// SIMATIC S7-200 project (STEP 7-Micro/WIN), CPU 224XP CN REL 02.01

SYMBOL_TABLE S7-200 符号
Always_On        SM0.0    // 始终接通为 ON
First_Scan_On    SM0.1    // 仅第一个扫描周期中接通为 ON
Xmit0_Idle       SM4.5    // 当发送器处于空闲状态时（端口 0），置位为 1
P0_Config        SMB30    // 通信端口 0 设置：奇偶校验、每个字符的数据位数目、波特率和协议
P0_Stat_Rcv      SMB86    // 端口 0 信息接收状态
P0_Ctrl_Rcv      SMB87    // 信息接收控制
P0_Start_Char    SMB88    // 信息起始字符
P0_End_Char      SMB89    // 信息结束字符
P0_Max_Char      SMB94    // 信息接收最大字符数（1 至 255 个字节）
P1_Config        SMB130   // 通信端口 1 设置：奇偶校验、每个字符的数据位数目、波特率和协议
P0_Idle_Time     SMW90    // 空闲线时间，以毫秒为单位表示
END_SYMBOL_TABLE

ORGANIZATION_BLOCK 主程序:OB1
TITLE=程序注释
BEGIN
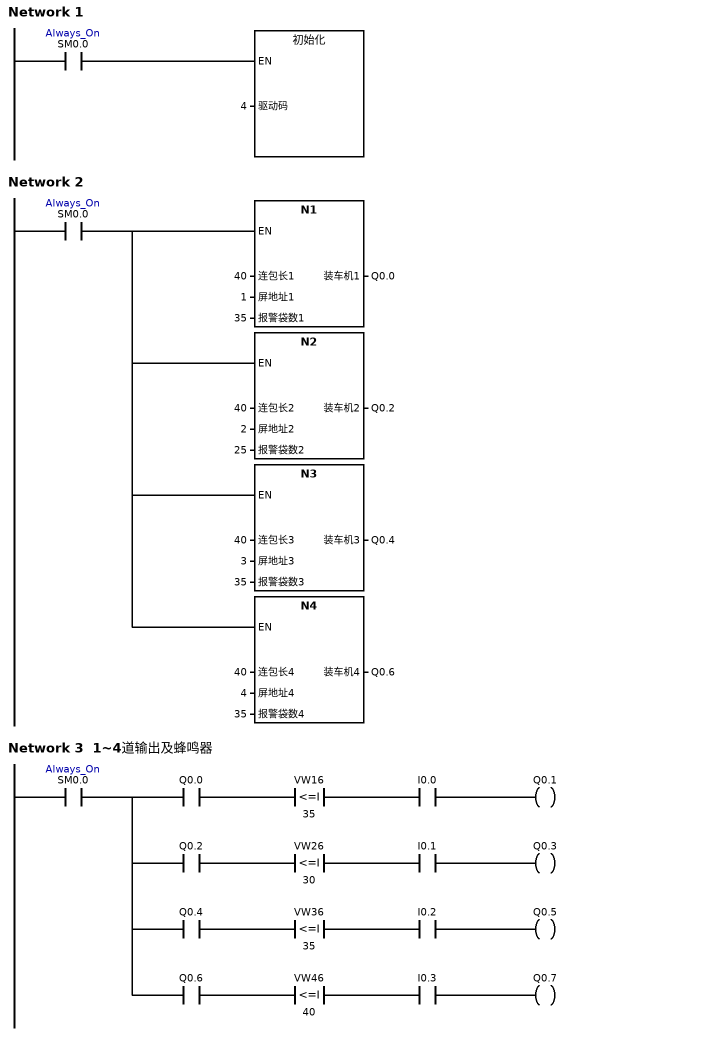
Network 1
LD     Always_On:SM0.0
CALL   初始化:SBR0, 4
Network 2
LD     Always_On:SM0.0
CALL   N1:SBR1, 40, 1, 35, Q0.0
CALL   N2:SBR2, 40, 2, 25, Q0.2
CALL   N3:SBR3, 40, 3, 35, Q0.4
CALL   N4:SBR4, 40, 4, 35, Q0.6
Network 3 // 1~4道输出及蜂鸣器
LD     Always_On:SM0.0
LPS
A      Q0.0
AW<=   VW16, 35
A      I0.0
=      Q0.1
LRD
A      Q0.2
AW<=   VW26, 30
A      I0.1
=      Q0.3
LRD
A      Q0.4
AW<=   VW36, 35
A      I0.2
=      Q0.5
LPP
A      Q0.6
AW<=   VW46, 40
A      I0.3
=      Q0.7
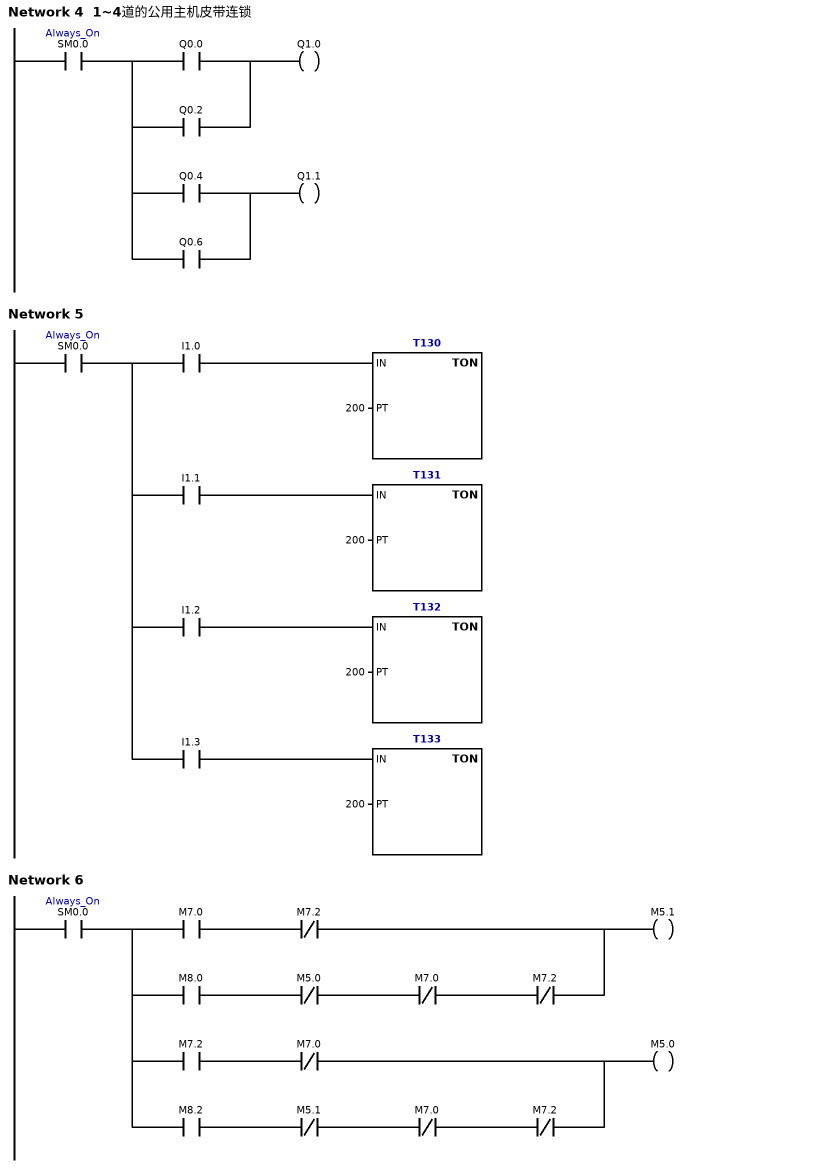
Network 4 // 1~4道的公用主机皮带连锁
LD     Always_On:SM0.0
LPS
LD     Q0.0
O      Q0.2
ALD
=      Q1.0
LPP
LD     Q0.4
O      Q0.6
ALD
=      Q1.1
Network 5
LD     Always_On:SM0.0
LPS
A      I1.0
TON    T130, 200
LRD
A      I1.1
TON    T131, 200
LRD
A      I1.2
TON    T132, 200
LPP
A      I1.3
TON    T133, 200
Network 6
LD     Always_On:SM0.0
LPS
LD     M7.0
AN     M7.2
LD     M8.0
AN     M5.0
AN     M7.0
AN     M7.2
OLD
ALD
=      M5.1
LPP
LD     M7.2
AN     M7.0
LD     M8.2
AN     M5.1
AN     M7.0
AN     M7.2
OLD
ALD
=      M5.0
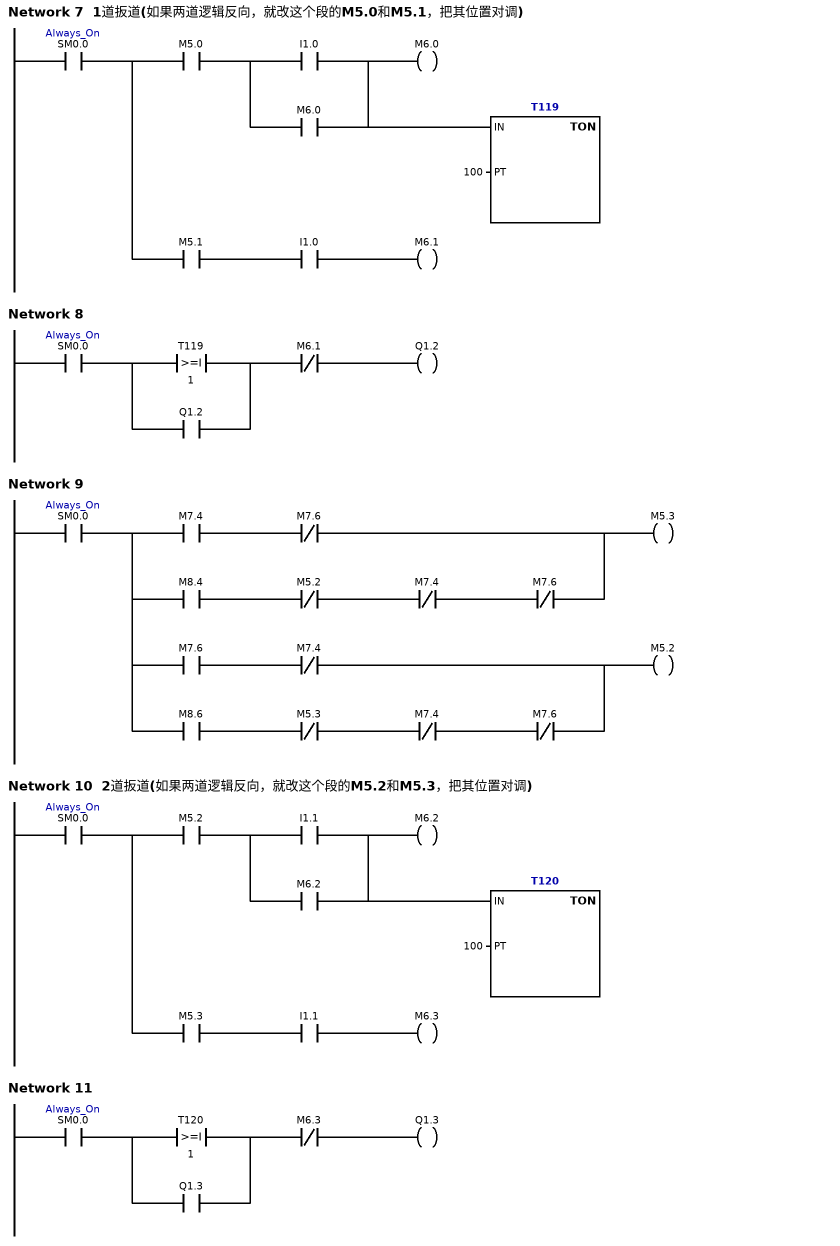
Network 7 // 1道扳道(如果两道逻辑反向，就改这个段的M5.0和M5.1，把其位置对调)
LD     Always_On:SM0.0
LPS
A      M5.0
LD     I1.0
O      M6.0
ALD
=      M6.0
TON    T119, 100
LPP
A      M5.1
A      I1.0
=      M6.1
Network 8
LD     Always_On:SM0.0
LDW>=  T119, 1
O      Q1.2
ALD
AN     M6.1
=      Q1.2
Network 9
LD     Always_On:SM0.0
LPS
LD     M7.4
AN     M7.6
LD     M8.4
AN     M5.2
AN     M7.4
AN     M7.6
OLD
ALD
=      M5.3
LPP
LD     M7.6
AN     M7.4
LD     M8.6
AN     M5.3
AN     M7.4
AN     M7.6
OLD
ALD
=      M5.2
Network 10 // 2道扳道(如果两道逻辑反向，就改这个段的M5.2和M5.3，把其位置对调)
LD     Always_On:SM0.0
LPS
A      M5.2
LD     I1.1
O      M6.2
ALD
=      M6.2
TON    T120, 100
LPP
A      M5.3
A      I1.1
=      M6.3
Network 11
LD     Always_On:SM0.0
LDW>=  T120, 1
O      Q1.3
ALD
AN     M6.3
=      Q1.3
END_ORGANIZATION_BLOCK

SUBROUTINE_BLOCK 初始化:SBR0
TITLE=子程序注释
VAR_INPUT
驱动码:WORD;	// LW0 
END_VAR
VAR
temp1:WORD;	// LW2 
temp2:WORD;	// LW4 
END_VAR
BEGIN
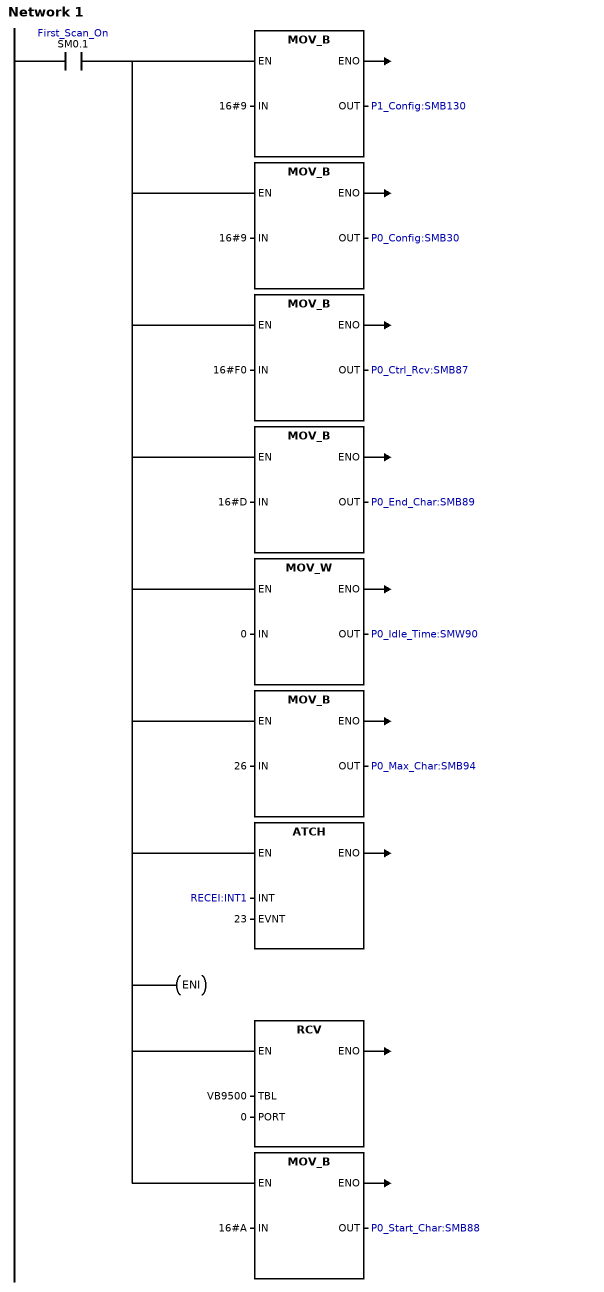
Network 1
// 首次扫描时，
// 初始化自由端口：
// - 选择9600波特
// - 选择8个数据位
// - 选择无校验
// 初始化RCV信息控制字节：
// - RCV被启用
// - 检测到信息字符结束
// - 将空闲行条件检测为
// 信息开始条件。
// 将信息字符结束设为hex OA（换行符）。
// 将空闲行超时设为5毫秒。
// 将最大字符数设为100。
// 为端口0在VB100位置启用带缓冲区的接收方框
LD     First_Scan_On:SM0.1
MOVB   16#9, P1_Config:SMB130
MOVB   16#9, P0_Config:SMB30
MOVB   16#F0, P0_Ctrl_Rcv:SMB87
MOVB   16#D, P0_End_Char:SMB89
MOVW   0, P0_Idle_Time:SMW90
MOVB   26, P0_Max_Char:SMB94
ATCH   RECEI:INT1, 23
ENI
RCV    VB9500, 0
MOVB   16#A, P0_Start_Char:SMB88
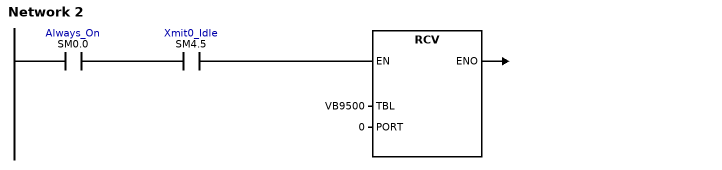
Network 2
LD     Always_On:SM0.0
A      Xmit0_Idle:SM4.5
RCV    VB9500, 0
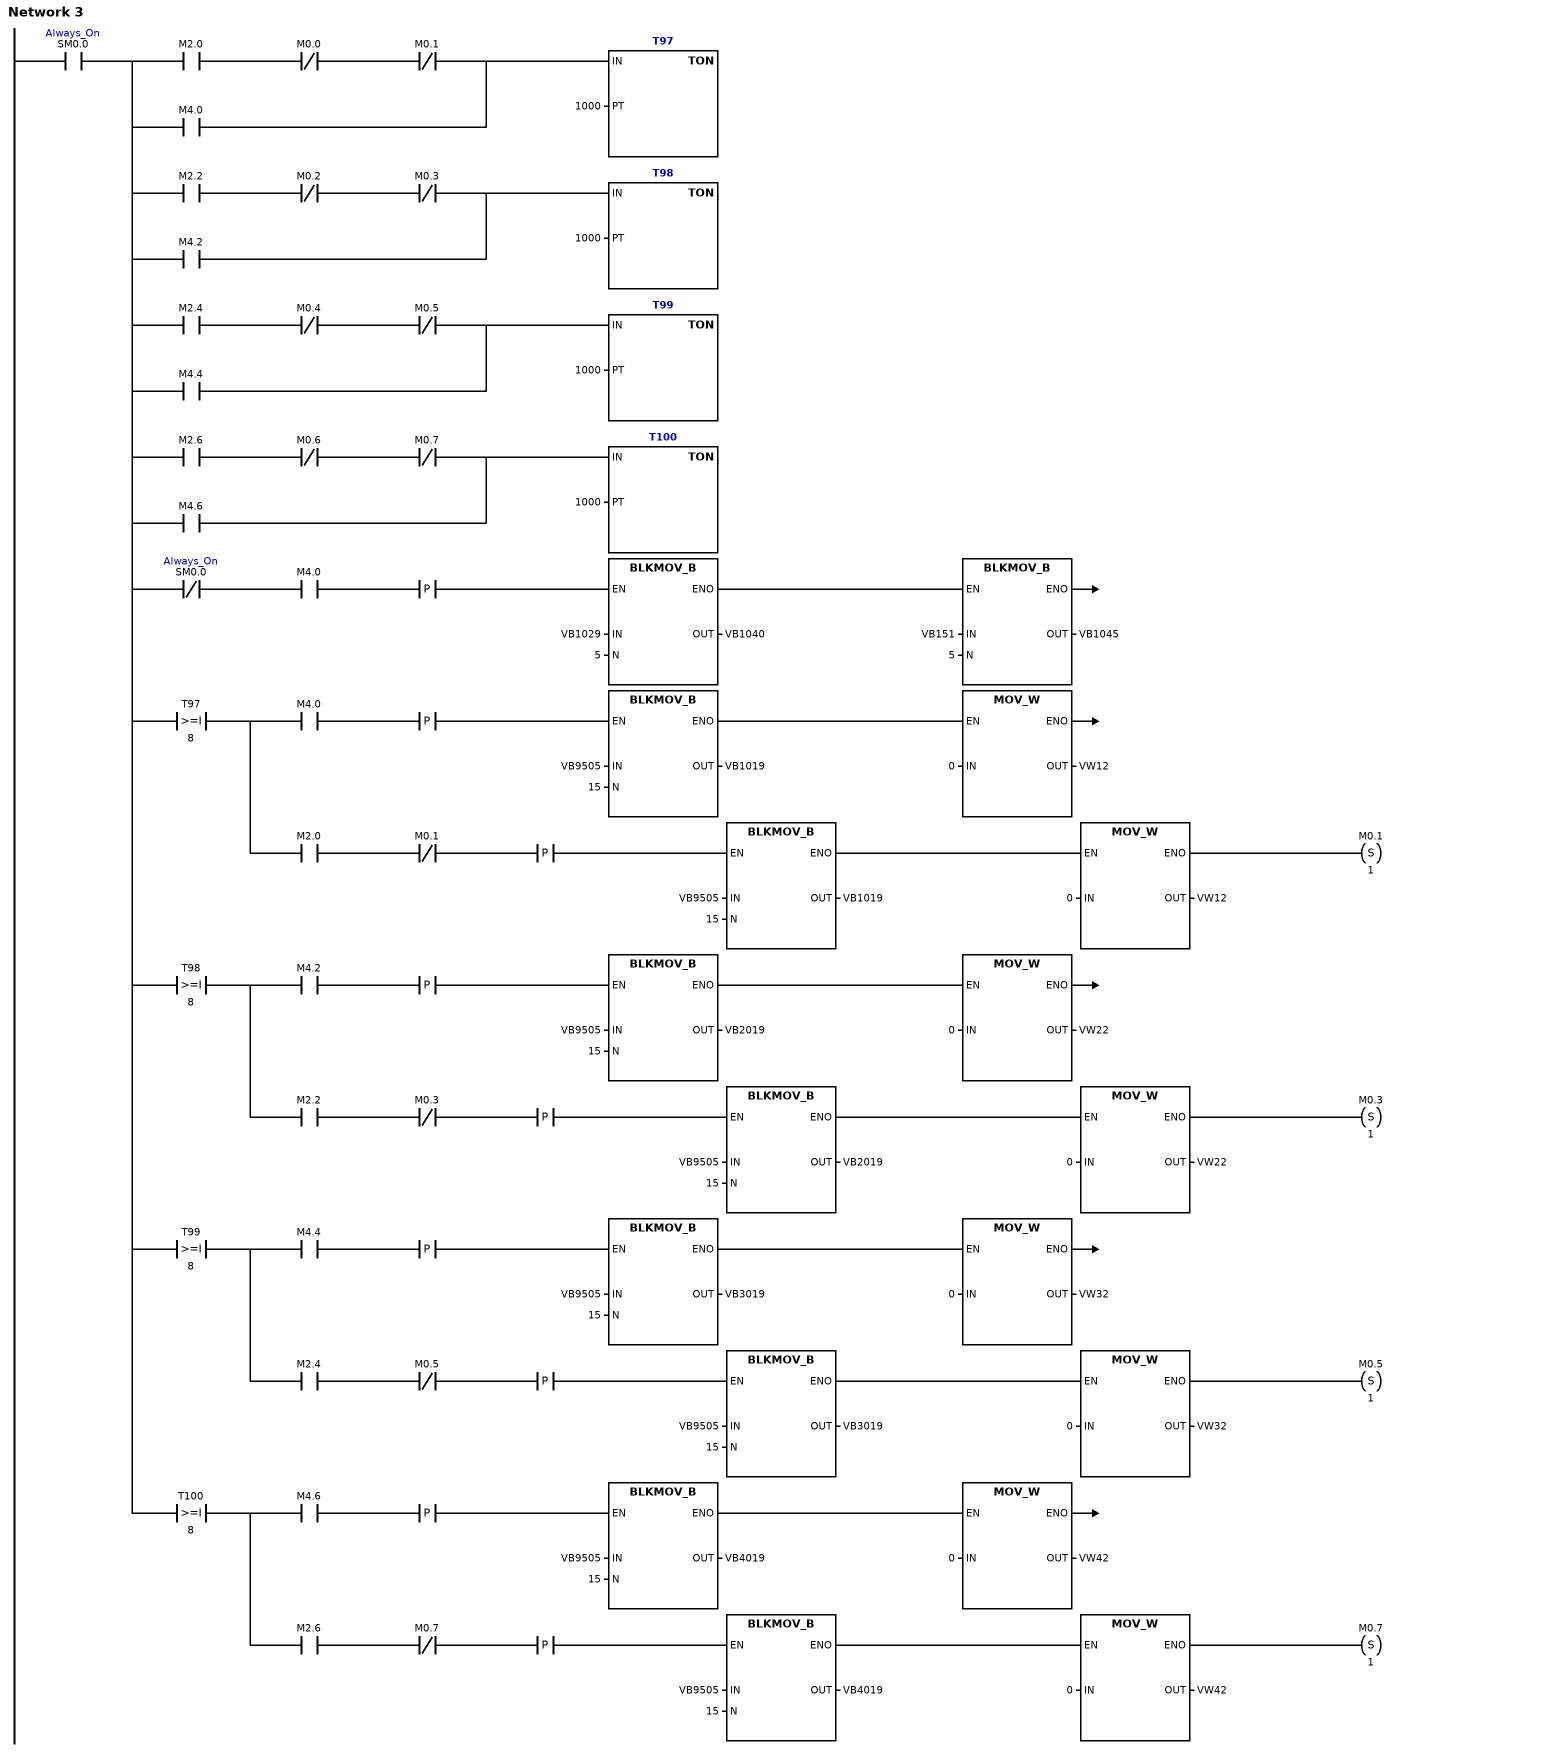
Network 3
LD     Always_On:SM0.0
LPS
LD     M2.0
AN     M0.0
AN     M0.1
O      M4.0
ALD
TON    T97, 1000
LRD
LD     M2.2
AN     M0.2
AN     M0.3
O      M4.2
ALD
TON    T98, 1000
LRD
LD     M2.4
AN     M0.4
AN     M0.5
O      M4.4
ALD
TON    T99, 1000
LRD
LD     M2.6
AN     M0.6
AN     M0.7
O      M4.6
ALD
TON    T100, 1000
LRD
AN     Always_On:SM0.0
A      M4.0
EU
BMB    VB1029, VB1040, 5
AENO
BMB    VB151, VB1045, 5
LRD
AW>=   T97, 8
LPS
A      M4.0
EU
BMB    VB9505, VB1019, 15
AENO
MOVW   0, VW12
LPP
A      M2.0
AN     M0.1
EU
BMB    VB9505, VB1019, 15
AENO
MOVW   0, VW12
AENO
S      M0.1, 1
LRD
AW>=   T98, 8
LPS
A      M4.2
EU
BMB    VB9505, VB2019, 15
AENO
MOVW   0, VW22
LPP
A      M2.2
AN     M0.3
EU
BMB    VB9505, VB2019, 15
AENO
MOVW   0, VW22
AENO
S      M0.3, 1
LRD
AW>=   T99, 8
LPS
A      M4.4
EU
BMB    VB9505, VB3019, 15
AENO
MOVW   0, VW32
LPP
A      M2.4
AN     M0.5
EU
BMB    VB9505, VB3019, 15
AENO
MOVW   0, VW32
AENO
S      M0.5, 1
LPP
AW>=   T100, 8
LPS
A      M4.6
EU
BMB    VB9505, VB4019, 15
AENO
MOVW   0, VW42
LPP
A      M2.6
AN     M0.7
EU
BMB    VB9505, VB4019, 15
AENO
MOVW   0, VW42
AENO
S      M0.7, 1
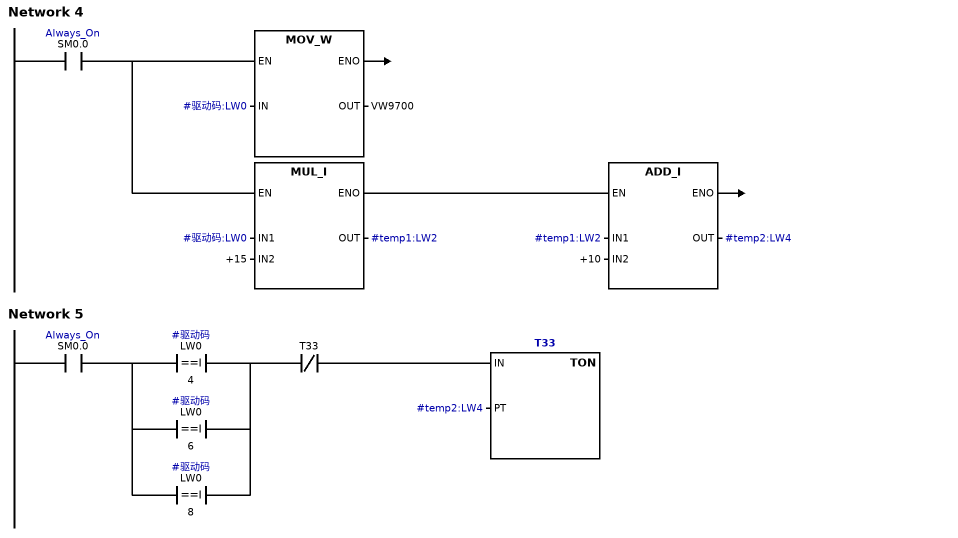
Network 4
LD     Always_On:SM0.0
MOVW   #驱动码:LW0, VW9700
MOVW   #驱动码:LW0, #temp1:LW2
AENO
*I     +15, #temp1:LW2
AENO
MOVW   #temp1:LW2, #temp2:LW4
+I     +10, #temp2:LW4
Network 5
LD     Always_On:SM0.0
LDW=   #驱动码:LW0, 4
OW=    #驱动码:LW0, 6
OW=    #驱动码:LW0, 8
ALD
AN     T33
TON    T33, #temp2:LW4
END_SUBROUTINE_BLOCK

SUBROUTINE_BLOCK N1:SBR1
TITLE=
VAR_INPUT
连包长1:WORD;	// LW0 
屏地址1:BYTE;	// LB2 
报警袋数1:WORD;	// LW3 
END_VAR
VAR_OUTPUT
装车机1:BOOL;	// L5.0 
END_VAR
VAR
总袋数1:WORD;	// LW6 
袋长1:WORD;	// LW8 
已装袋数1:WORD;	// LW10 
剩余袋数1:WORD;	// LW12 
END_VAR
BEGIN
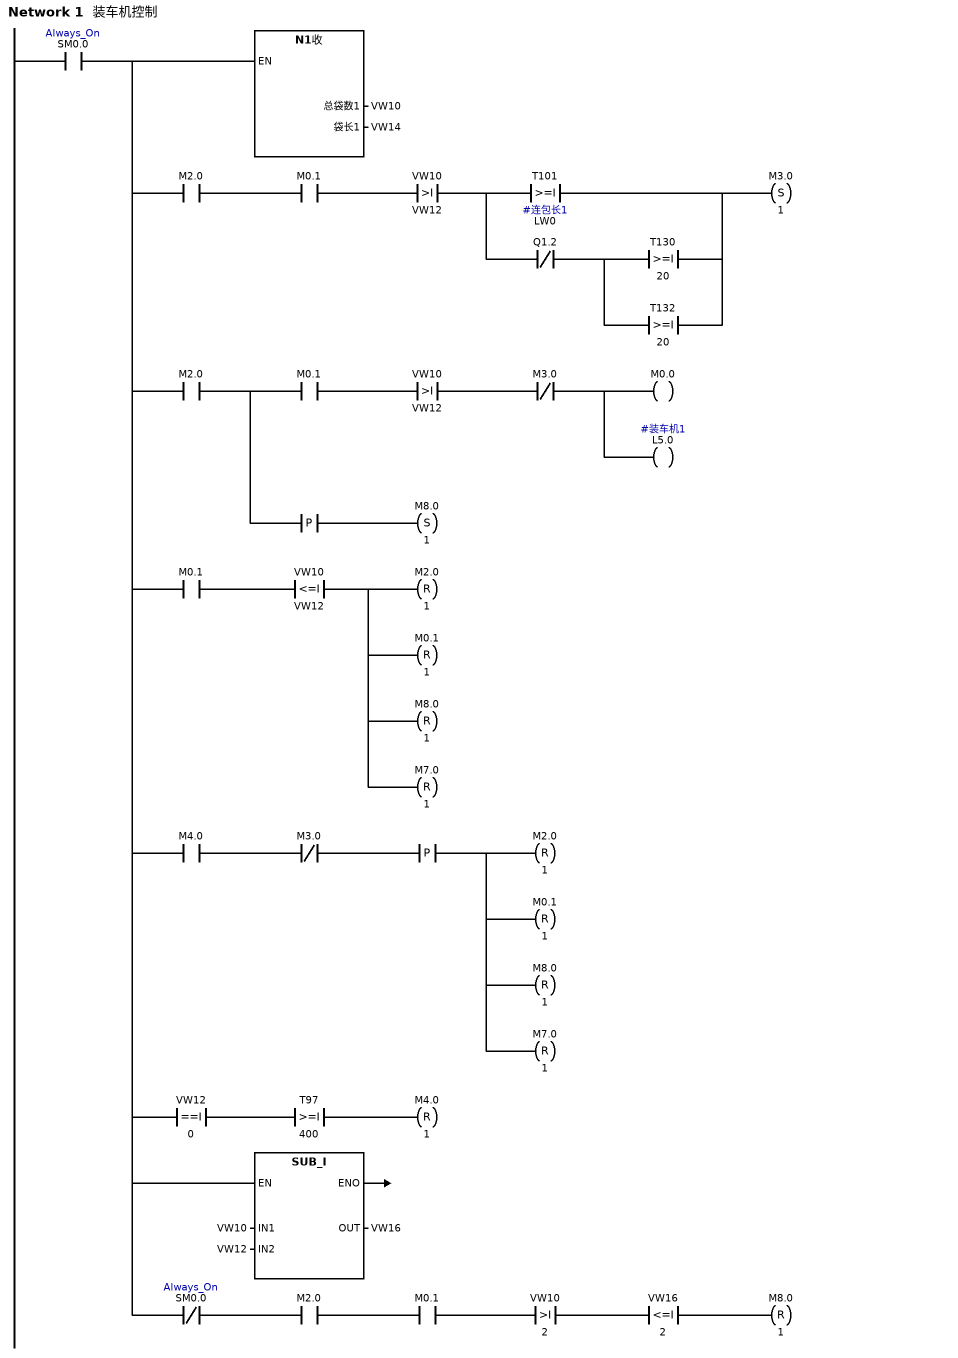
Network 1 // 装车机控制
LD     Always_On:SM0.0
LPS
CALL   N1收:SBR21, VW10, VW14
A      M2.0
A      M0.1
AW>    VW10, VW12
LDW>=  T101, #连包长1:LW0
LDN    Q1.2
LDW>=  T130, 20
OW>=   T132, 20
ALD
OLD
ALD
S      M3.0, 1
LRD
A      M2.0
LPS
A      M0.1
AW>    VW10, VW12
AN     M3.0
=      M0.0
=      #装车机1:L5.0
LPP
EU
S      M8.0, 1
LPP
LPS
A      M0.1
AW<=   VW10, VW12
R      M2.0, 1
R      M0.1, 1
R      M8.0, 1
R      M7.0, 1
LRD
A      M4.0
AN     M3.0
EU
R      M2.0, 1
R      M0.1, 1
R      M8.0, 1
R      M7.0, 1
LPP
LPS
AW=    VW12, 0
AW>=   T97, 400
R      M4.0, 1
LRD
MOVW   VW10, VW16
-I     VW12, VW16
LPP
AN     Always_On:SM0.0
A      M2.0
A      M0.1
AW>    VW10, 2
AW<=   VW16, 2
R      M8.0, 1
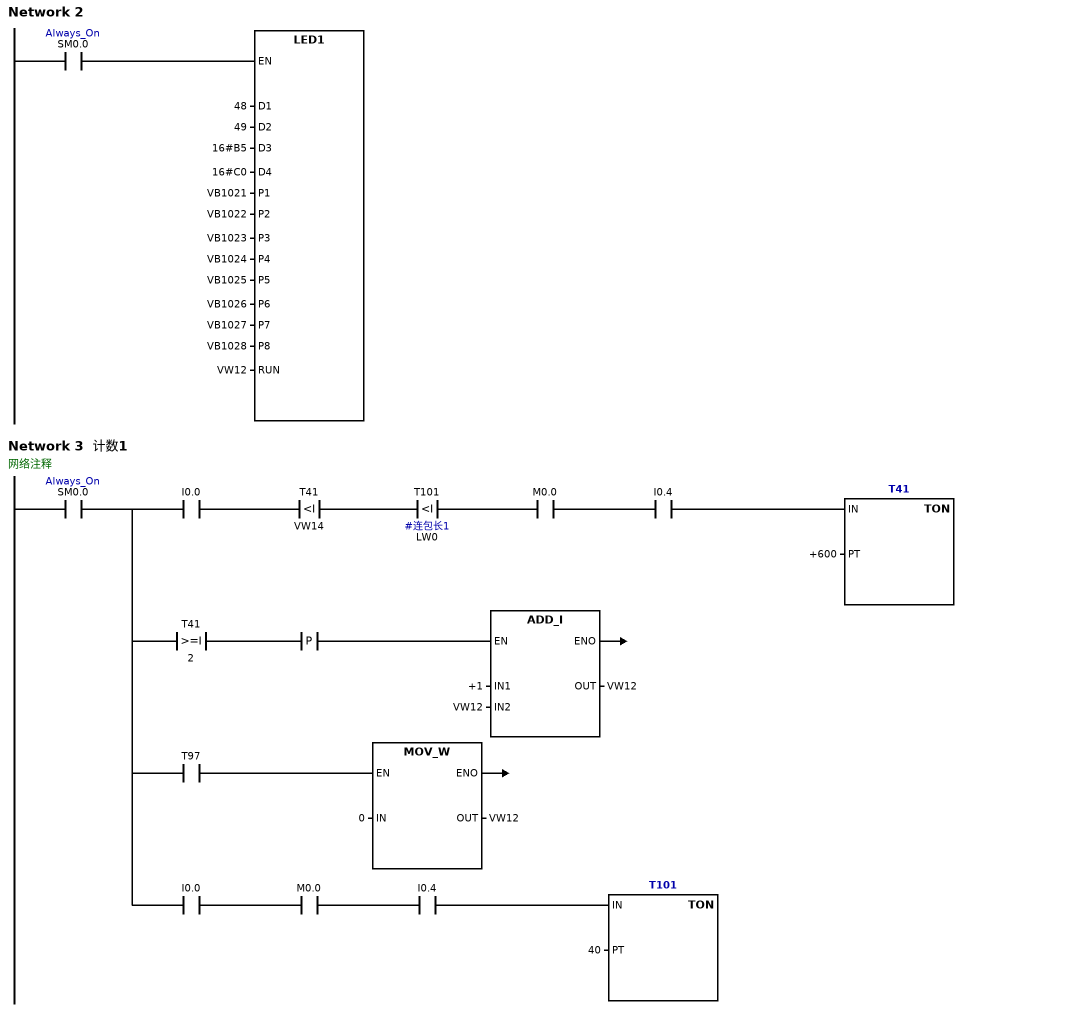
Network 2
LD     Always_On:SM0.0
CALL   LED1:SBR11, 48, 49, 16#B5, 16#C0, VB1021, VB1022, VB1023, VB1024, VB1025, VB1026, VB1027, VB1028, VW12
Network 3 // 计数1
// 网络注释
LD     Always_On:SM0.0
LPS
A      I0.0
AW<    T41, VW14
AW<    T101, #连包长1:LW0
A      M0.0
A      I0.4
TON    T41, +600
LRD
AW>=   T41, 2
EU
+I     +1, VW12
LRD
A      T97
MOVW   0, VW12
LPP
A      I0.0
A      M0.0
A      I0.4
TON    T101, 40
END_SUBROUTINE_BLOCK

SUBROUTINE_BLOCK N2:SBR2
TITLE=
VAR_INPUT
连包长2:WORD;	// LW0 
屏地址2:BYTE;	// LB2 
报警袋数2:WORD;	// LW3 
END_VAR
VAR_OUTPUT
装车机2:BOOL;	// L5.0 
END_VAR
VAR
总袋数2:WORD;	// LW6 
袋长2:WORD;	// LW8 
已装袋数2:WORD;	// LW10 
剩余袋数2:WORD;	// LW12 
END_VAR
BEGIN
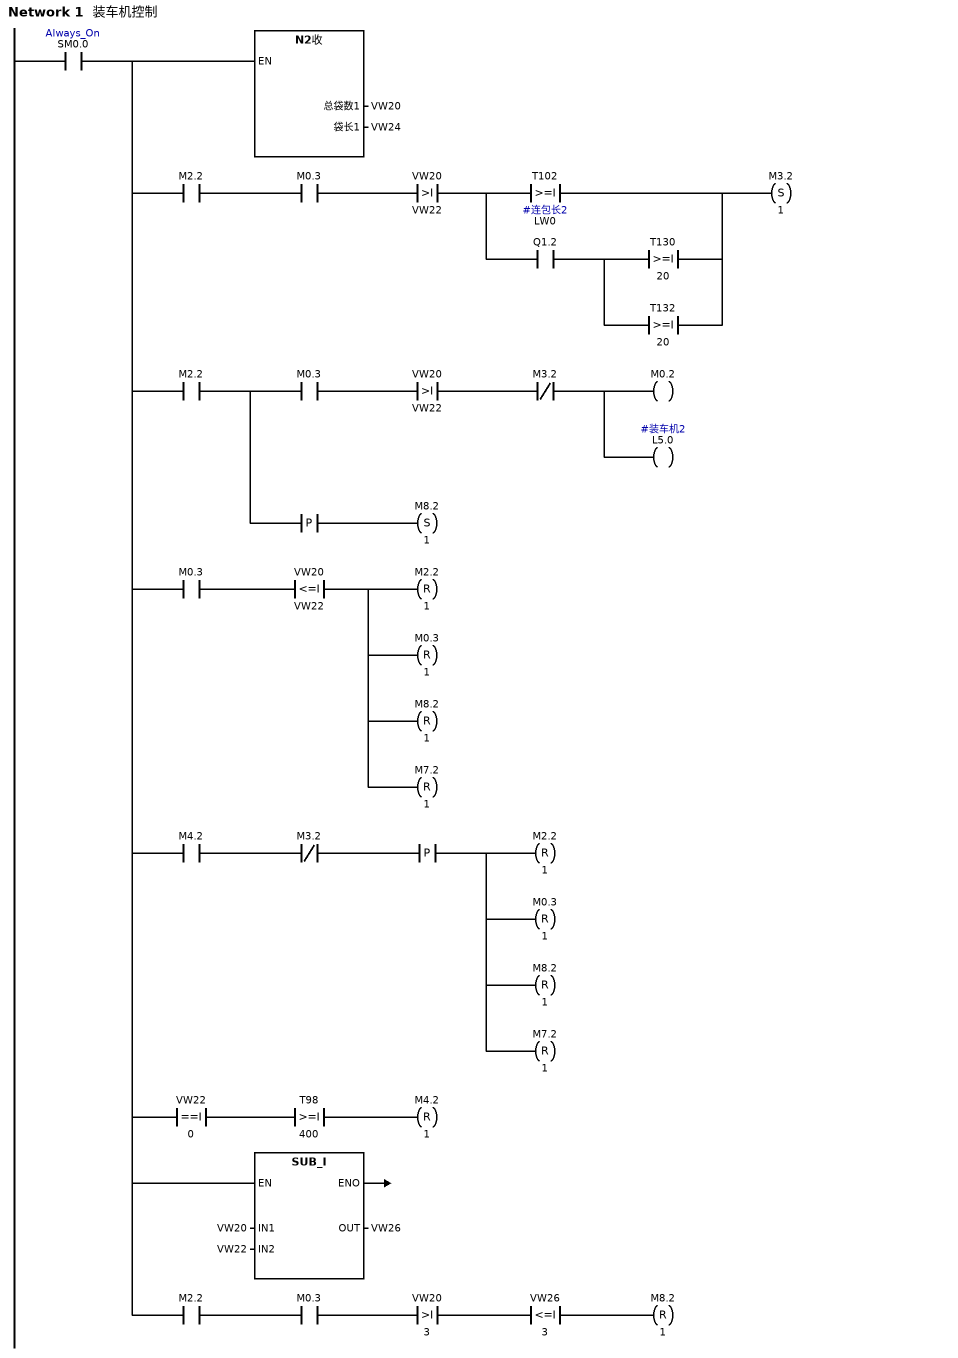
Network 1 // 装车机控制
LD     Always_On:SM0.0
LPS
CALL   N2收:SBR22, VW20, VW24
A      M2.2
A      M0.3
AW>    VW20, VW22
LDW>=  T102, #连包长2:LW0
LD     Q1.2
LDW>=  T130, 20
OW>=   T132, 20
ALD
OLD
ALD
S      M3.2, 1
LRD
A      M2.2
LPS
A      M0.3
AW>    VW20, VW22
AN     M3.2
=      M0.2
=      #装车机2:L5.0
LPP
EU
S      M8.2, 1
LPP
LPS
A      M0.3
AW<=   VW20, VW22
R      M2.2, 1
R      M0.3, 1
R      M8.2, 1
R      M7.2, 1
LRD
A      M4.2
AN     M3.2
EU
R      M2.2, 1
R      M0.3, 1
R      M8.2, 1
R      M7.2, 1
LPP
LPS
AW=    VW22, 0
AW>=   T98, 400
R      M4.2, 1
LRD
MOVW   VW20, VW26
-I     VW22, VW26
LPP
A      M2.2
A      M0.3
AW>    VW20, 3
AW<=   VW26, 3
R      M8.2, 1
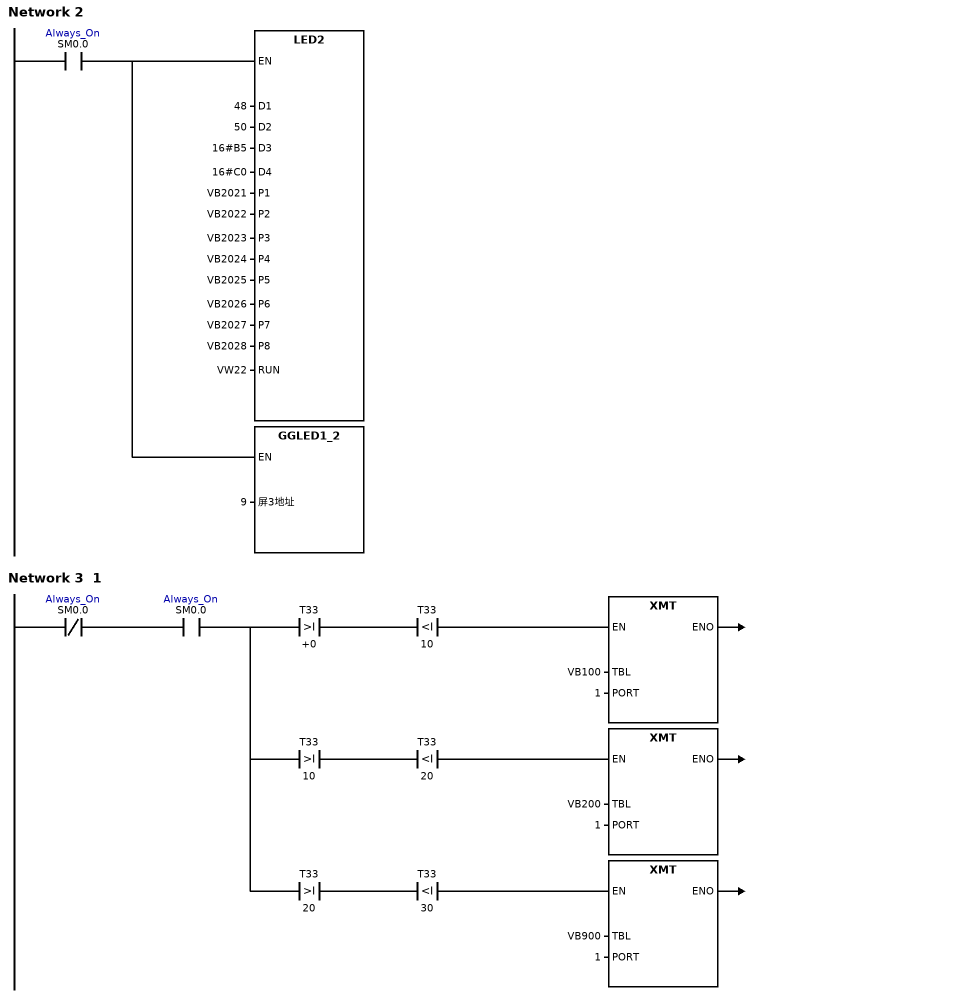
Network 2
LD     Always_On:SM0.0
CALL   LED2:SBR12, 48, 50, 16#B5, 16#C0, VB2021, VB2022, VB2023, VB2024, VB2025, VB2026, VB2027, VB2028, VW22
CALL   GGLED1_2:SBR31, 9
Network 3 // 1
LDN    Always_On:SM0.0
A      Always_On:SM0.0
LPS
AW>    T33, +0
AW<    T33, 10
XMT    VB100, 1
LRD
AW>    T33, 10
AW<    T33, 20
XMT    VB200, 1
LPP
AW>    T33, 20
AW<    T33, 30
XMT    VB900, 1
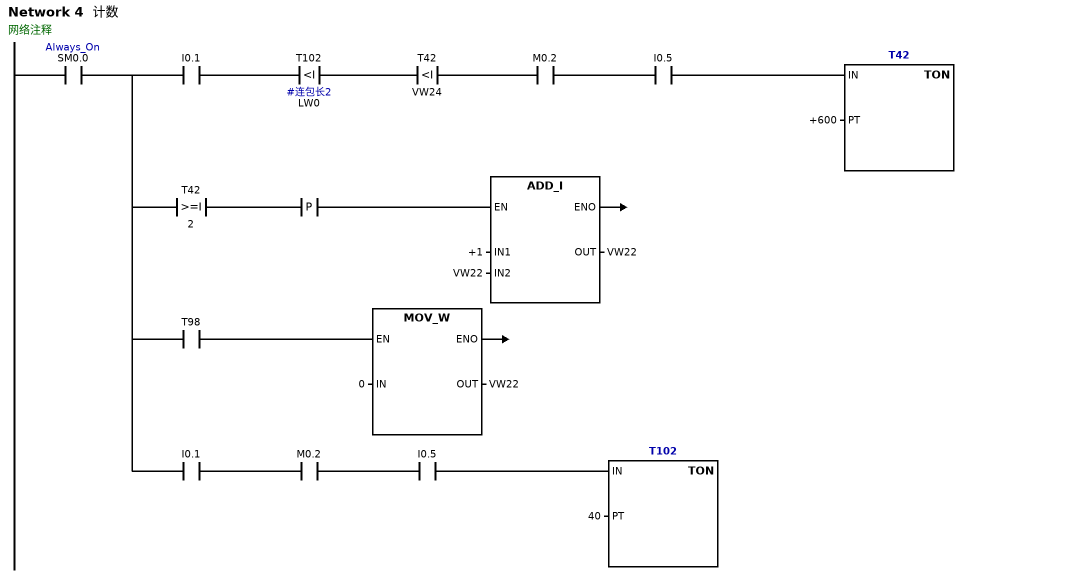
Network 4 // 计数
// 网络注释
LD     Always_On:SM0.0
LPS
A      I0.1
AW<    T102, #连包长2:LW0
AW<    T42, VW24
A      M0.2
A      I0.5
TON    T42, +600
LRD
AW>=   T42, 2
EU
+I     +1, VW22
LRD
A      T98
MOVW   0, VW22
LPP
A      I0.1
A      M0.2
A      I0.5
TON    T102, 40
END_SUBROUTINE_BLOCK

SUBROUTINE_BLOCK N3:SBR3
TITLE=
VAR_INPUT
连包长3:WORD;	// LW0 
屏地址3:BYTE;	// LB2 
报警袋数3:WORD;	// LW3 
END_VAR
VAR_OUTPUT
装车机3:BOOL;	// L5.0 
END_VAR
VAR
总袋数3:WORD;	// LW6 
袋长3:WORD;	// LW8 
已装袋数3:WORD;	// LW10 
剩余袋数3:WORD;	// LW12 
END_VAR
BEGIN
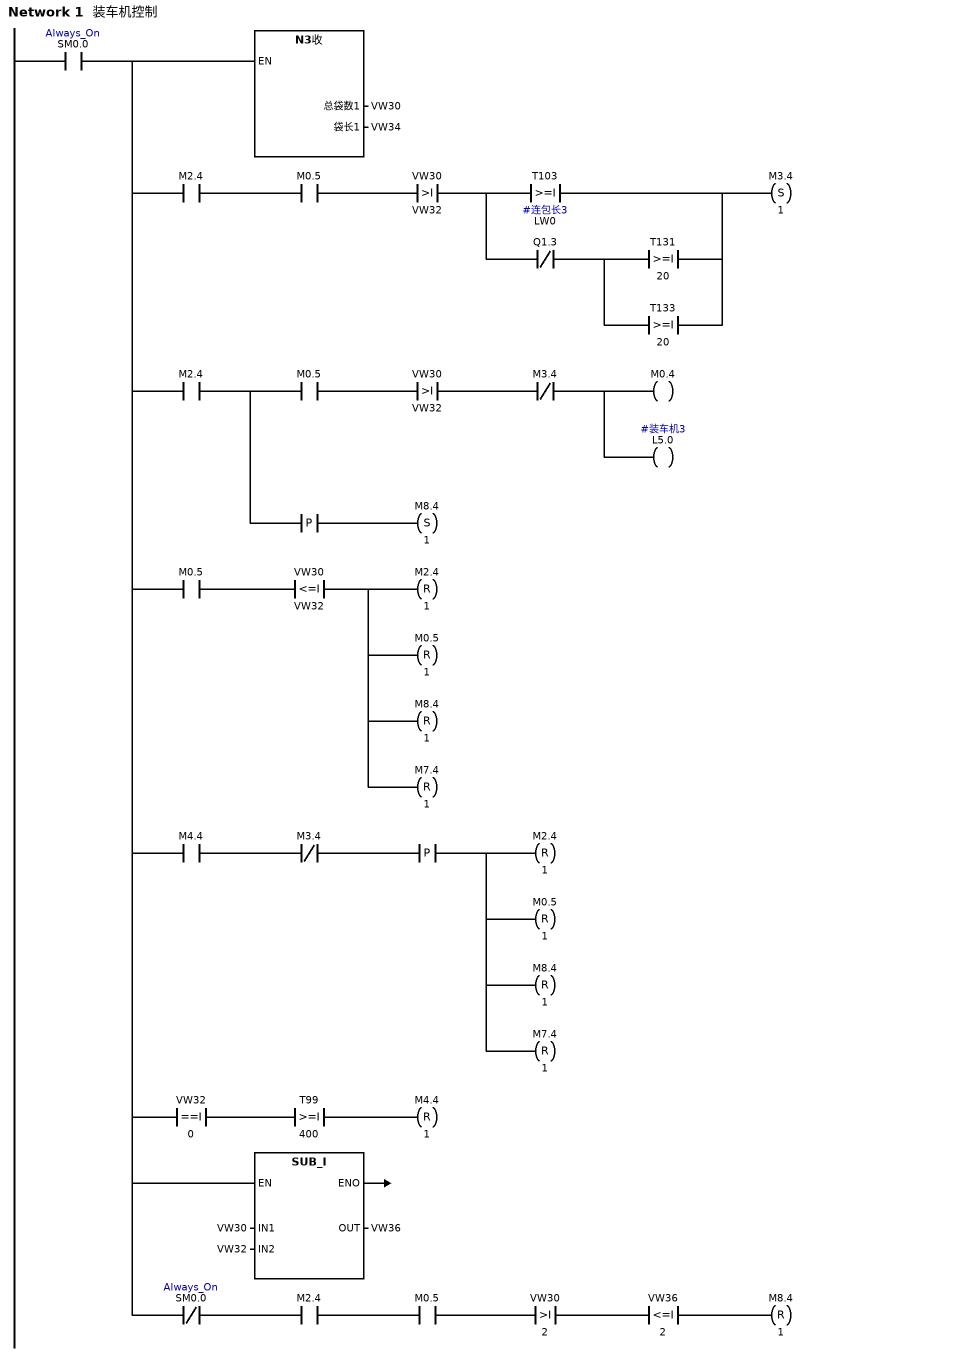
Network 1 // 装车机控制
LD     Always_On:SM0.0
LPS
CALL   N3收:SBR23, VW30, VW34
A      M2.4
A      M0.5
AW>    VW30, VW32
LDW>=  T103, #连包长3:LW0
LDN    Q1.3
LDW>=  T131, 20
OW>=   T133, 20
ALD
OLD
ALD
S      M3.4, 1
LRD
A      M2.4
LPS
A      M0.5
AW>    VW30, VW32
AN     M3.4
=      M0.4
=      #装车机3:L5.0
LPP
EU
S      M8.4, 1
LPP
LPS
A      M0.5
AW<=   VW30, VW32
R      M2.4, 1
R      M0.5, 1
R      M8.4, 1
R      M7.4, 1
LRD
A      M4.4
AN     M3.4
EU
R      M2.4, 1
R      M0.5, 1
R      M8.4, 1
R      M7.4, 1
LPP
LPS
AW=    VW32, 0
AW>=   T99, 400
R      M4.4, 1
LRD
MOVW   VW30, VW36
-I     VW32, VW36
LPP
AN     Always_On:SM0.0
A      M2.4
A      M0.5
AW>    VW30, 2
AW<=   VW36, 2
R      M8.4, 1
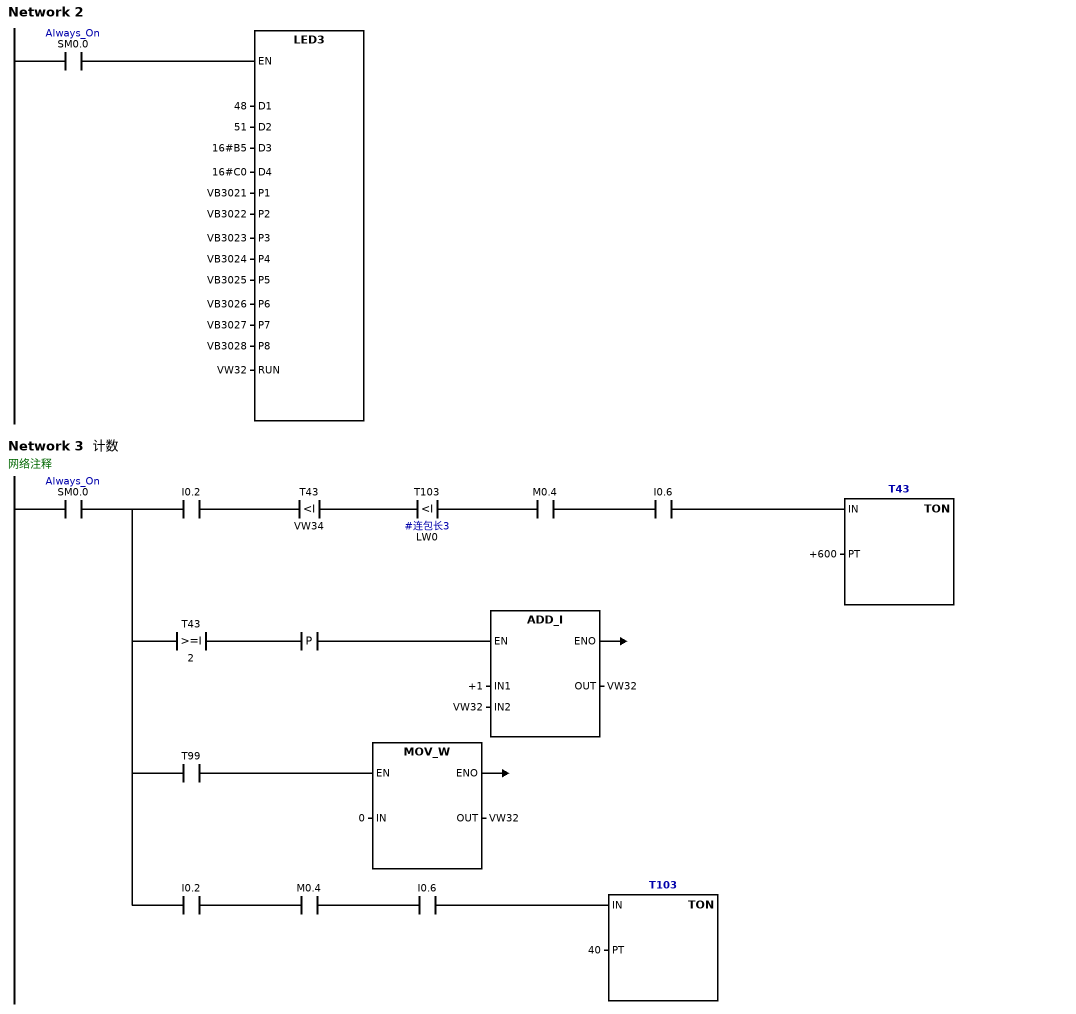
Network 2
LD     Always_On:SM0.0
CALL   LED3:SBR13, 48, 51, 16#B5, 16#C0, VB3021, VB3022, VB3023, VB3024, VB3025, VB3026, VB3027, VB3028, VW32
Network 3 // 计数
// 网络注释
LD     Always_On:SM0.0
LPS
A      I0.2
AW<    T43, VW34
AW<    T103, #连包长3:LW0
A      M0.4
A      I0.6
TON    T43, +600
LRD
AW>=   T43, 2
EU
+I     +1, VW32
LRD
A      T99
MOVW   0, VW32
LPP
A      I0.2
A      M0.4
A      I0.6
TON    T103, 40
END_SUBROUTINE_BLOCK

SUBROUTINE_BLOCK N4:SBR4
TITLE=
VAR_INPUT
连包长4:WORD;	// LW0 
屏地址4:BYTE;	// LB2 
报警袋数4:WORD;	// LW3 
END_VAR
VAR_OUTPUT
装车机4:BOOL;	// L5.0 
END_VAR
VAR
总袋数4:WORD;	// LW6 
袋长4:WORD;	// LW8 
已装袋数4:WORD;	// LW10 
剩余袋数4:WORD;	// LW12 
END_VAR
BEGIN
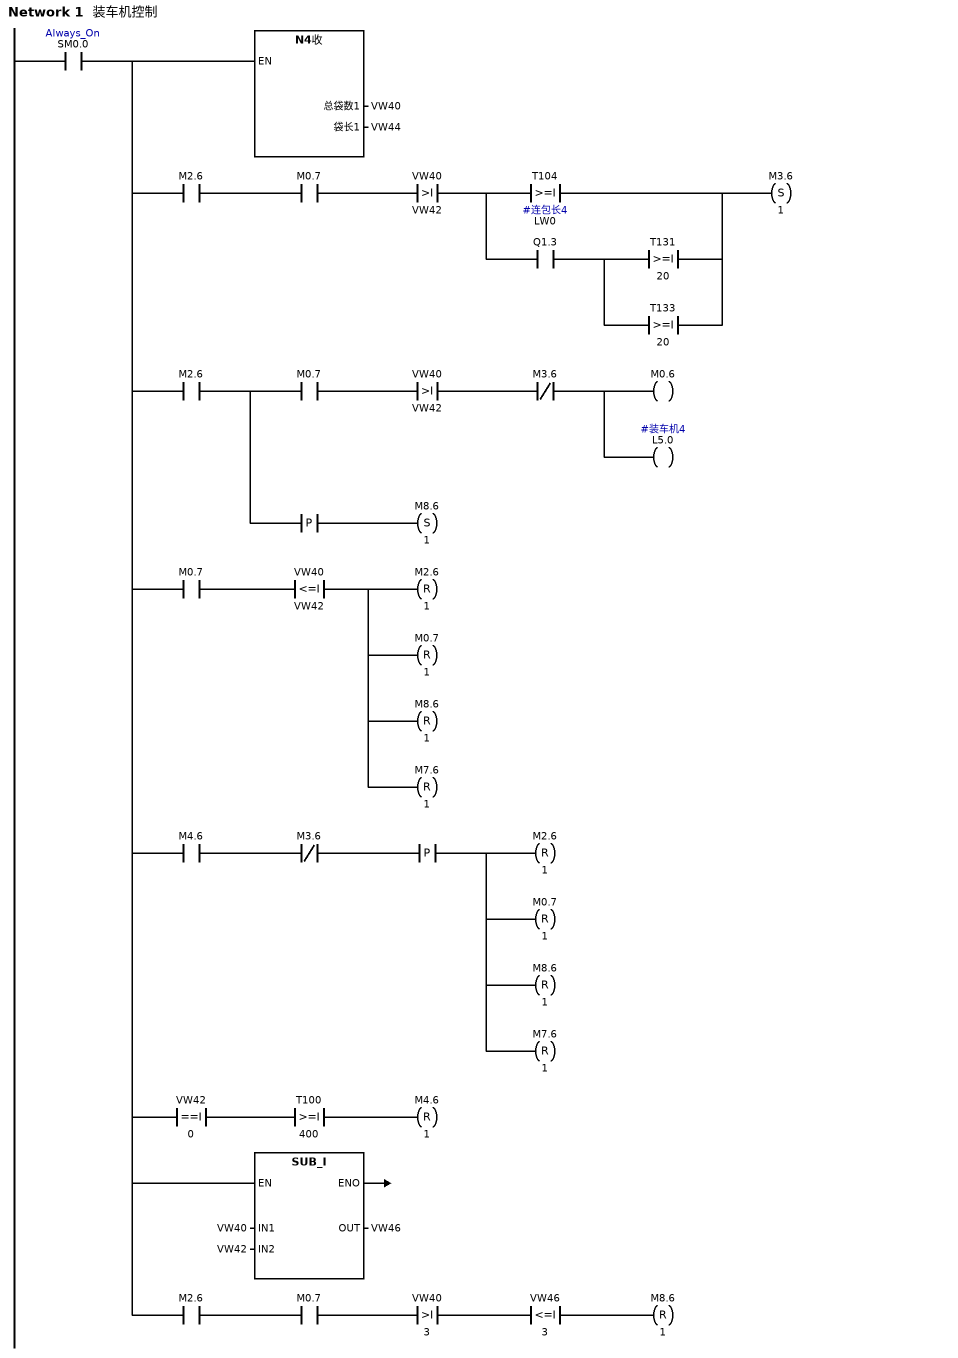
Network 1 // 装车机控制
LD     Always_On:SM0.0
LPS
CALL   N4收:SBR24, VW40, VW44
A      M2.6
A      M0.7
AW>    VW40, VW42
LDW>=  T104, #连包长4:LW0
LD     Q1.3
LDW>=  T131, 20
OW>=   T133, 20
ALD
OLD
ALD
S      M3.6, 1
LRD
A      M2.6
LPS
A      M0.7
AW>    VW40, VW42
AN     M3.6
=      M0.6
=      #装车机4:L5.0
LPP
EU
S      M8.6, 1
LPP
LPS
A      M0.7
AW<=   VW40, VW42
R      M2.6, 1
R      M0.7, 1
R      M8.6, 1
R      M7.6, 1
LRD
A      M4.6
AN     M3.6
EU
R      M2.6, 1
R      M0.7, 1
R      M8.6, 1
R      M7.6, 1
LPP
LPS
AW=    VW42, 0
AW>=   T100, 400
R      M4.6, 1
LRD
MOVW   VW40, VW46
-I     VW42, VW46
LPP
A      M2.6
A      M0.7
AW>    VW40, 3
AW<=   VW46, 3
R      M8.6, 1
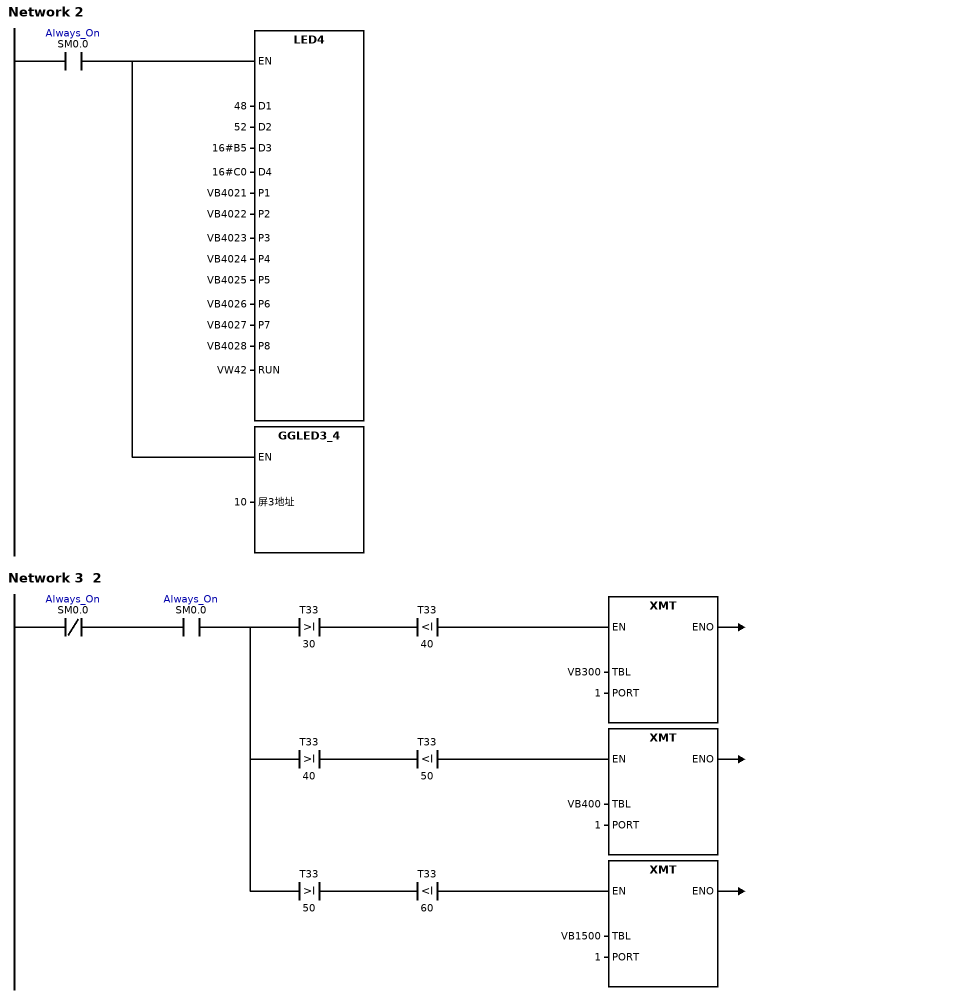
Network 2
LD     Always_On:SM0.0
CALL   LED4:SBR14, 48, 52, 16#B5, 16#C0, VB4021, VB4022, VB4023, VB4024, VB4025, VB4026, VB4027, VB4028, VW42
CALL   GGLED3_4:SBR32, 10
Network 3 // 2
LDN    Always_On:SM0.0
A      Always_On:SM0.0
LPS
AW>    T33, 30
AW<    T33, 40
XMT    VB300, 1
LRD
AW>    T33, 40
AW<    T33, 50
XMT    VB400, 1
LPP
AW>    T33, 50
AW<    T33, 60
XMT    VB1500, 1
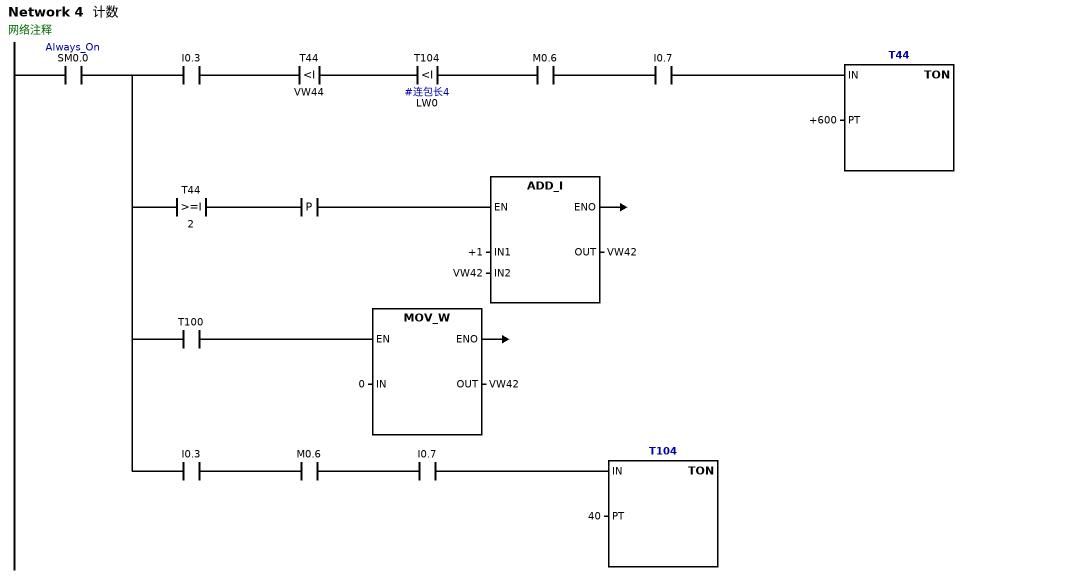
Network 4 // 计数
// 网络注释
LD     Always_On:SM0.0
LPS
A      I0.3
AW<    T44, VW44
AW<    T104, #连包长4:LW0
A      M0.6
A      I0.7
TON    T44, +600
LRD
AW>=   T44, 2
EU
+I     +1, VW42
LRD
A      T100
MOVW   0, VW42
LPP
A      I0.3
A      M0.6
A      I0.7
TON    T104, 40
END_SUBROUTINE_BLOCK

SUBROUTINE_BLOCK LED1:SBR11
TITLE=
VAR_INPUT
D1:BYTE;	// LB0 
D2:BYTE;	// LB1 
D3:BYTE;	// LB2 
D4:BYTE;	// LB3 
P1:BYTE;	// LB4 
P2:BYTE;	// LB5 
P3:BYTE;	// LB6 
P4:BYTE;	// LB7 
P5:BYTE;	// LB8 
P6:BYTE;	// LB9 
P7:BYTE;	// LB10 
P8:BYTE;	// LB11 
RUN:WORD;	// LW12 
END_VAR
BEGIN
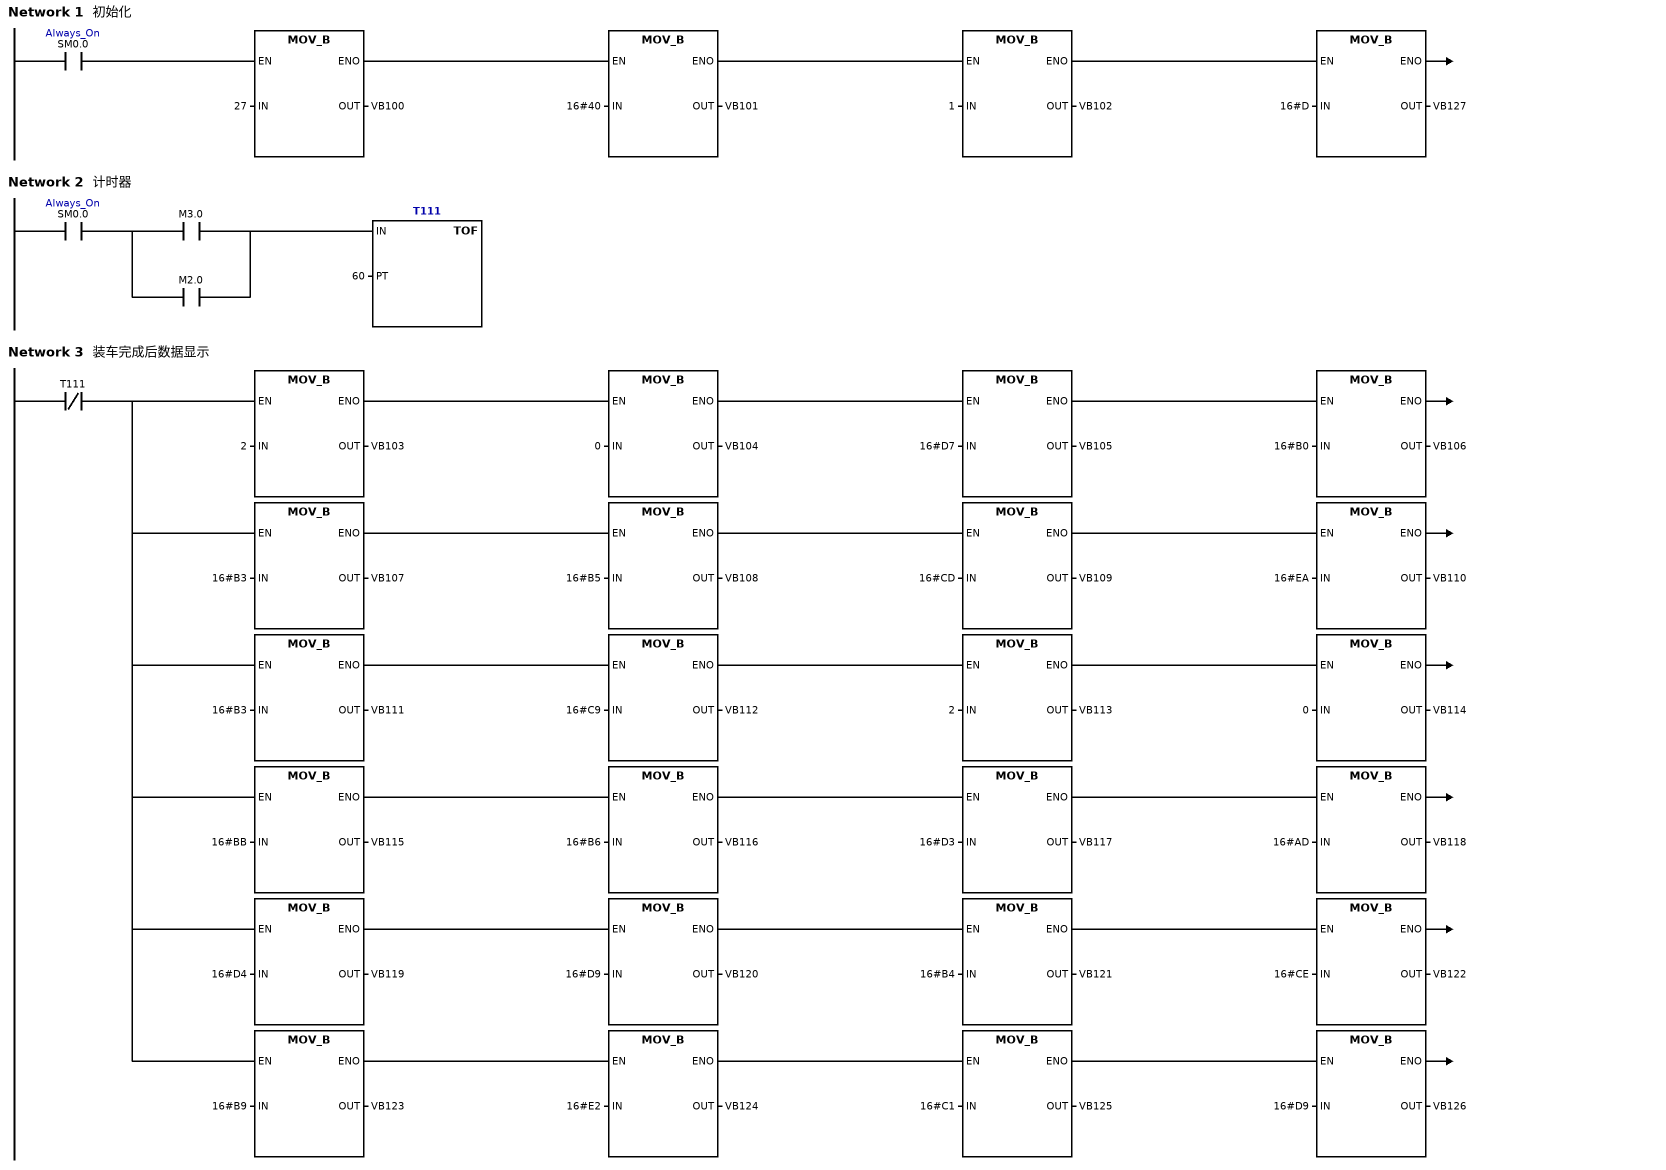
Network 1 // 初始化
LD     Always_On:SM0.0
MOVB   27, VB100
AENO
MOVB   16#40, VB101
AENO
MOVB   1, VB102
AENO
MOVB   16#D, VB127
Network 2 // 计时器
LD     Always_On:SM0.0
LD     M3.0
O      M2.0
ALD
TOF    T111, 60
Network 3 // 装车完成后数据显示
LDN    T111
LPS
MOVB   2, VB103
AENO
MOVB   0, VB104
AENO
MOVB   16#D7, VB105
AENO
MOVB   16#B0, VB106
LRD
MOVB   16#B3, VB107
AENO
MOVB   16#B5, VB108
AENO
MOVB   16#CD, VB109
AENO
MOVB   16#EA, VB110
LRD
MOVB   16#B3, VB111
AENO
MOVB   16#C9, VB112
AENO
MOVB   2, VB113
AENO
MOVB   0, VB114
LRD
MOVB   16#BB, VB115
AENO
MOVB   16#B6, VB116
AENO
MOVB   16#D3, VB117
AENO
MOVB   16#AD, VB118
LRD
MOVB   16#D4, VB119
AENO
MOVB   16#D9, VB120
AENO
MOVB   16#B4, VB121
AENO
MOVB   16#CE, VB122
LPP
MOVB   16#B9, VB123
AENO
MOVB   16#E2, VB124
AENO
MOVB   16#C1, VB125
AENO
MOVB   16#D9, VB126
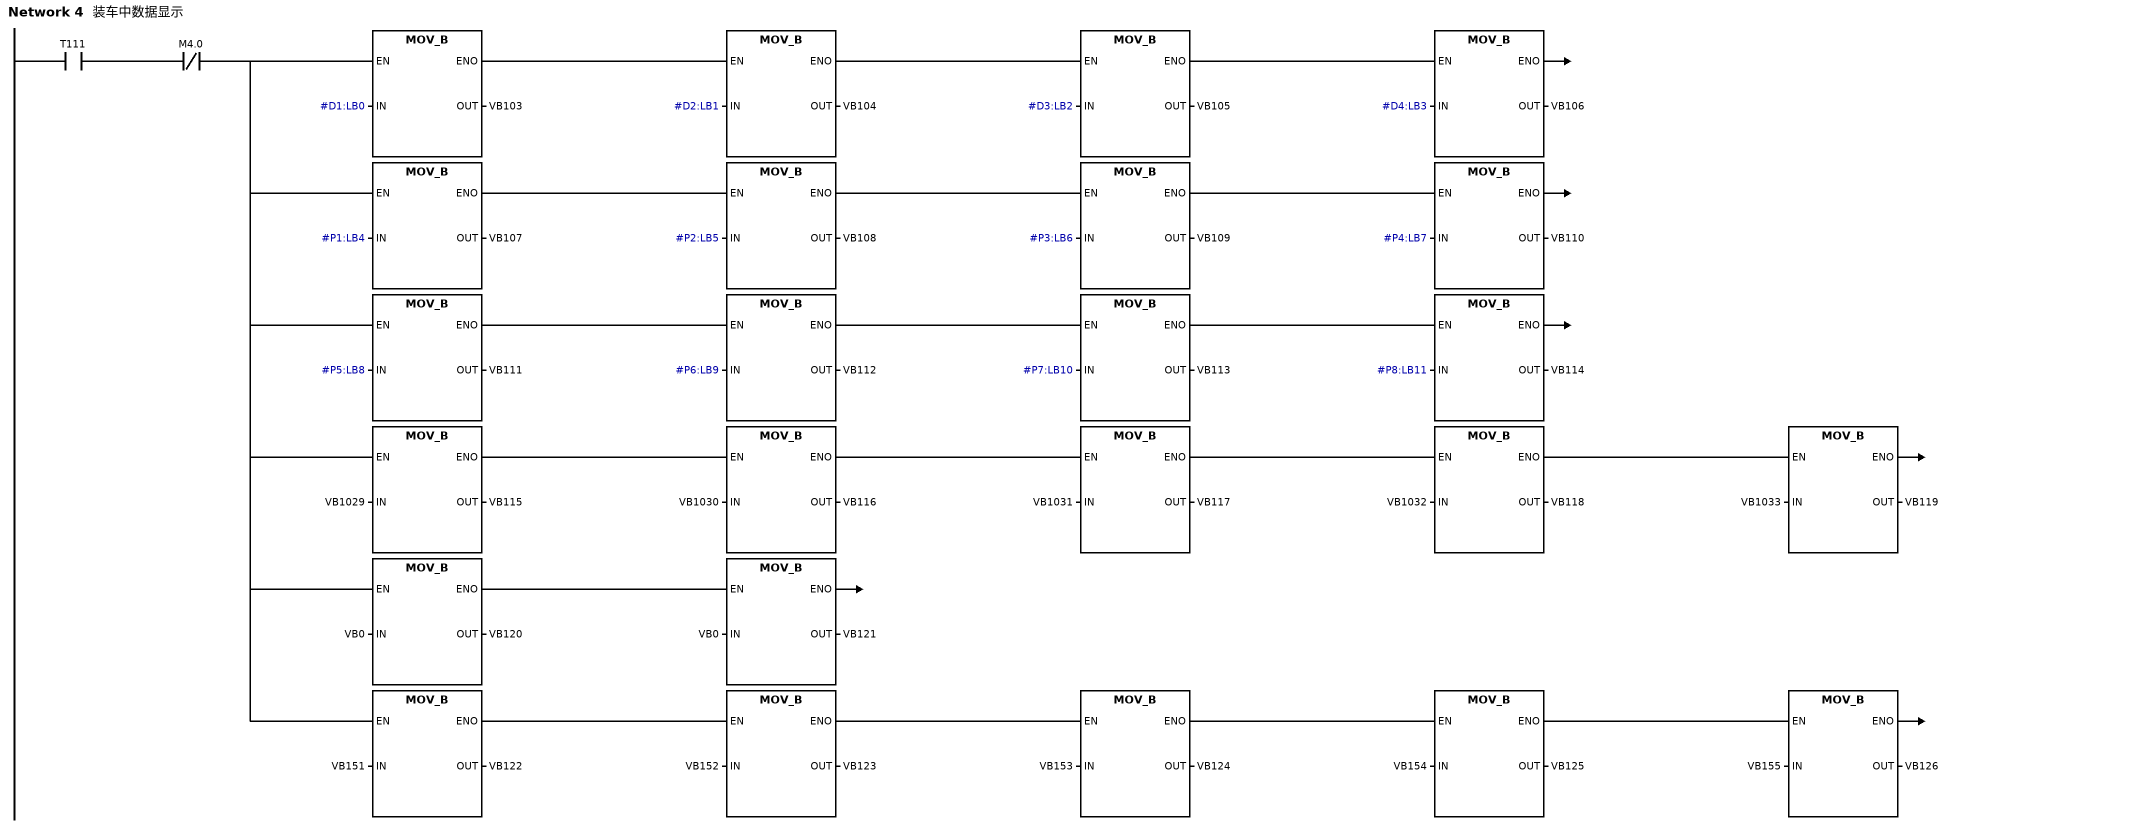
Network 4 // 装车中数据显示
LD     T111
AN     M4.0
LPS
MOVB   #D1:LB0, VB103
AENO
MOVB   #D2:LB1, VB104
AENO
MOVB   #D3:LB2, VB105
AENO
MOVB   #D4:LB3, VB106
LRD
MOVB   #P1:LB4, VB107
AENO
MOVB   #P2:LB5, VB108
AENO
MOVB   #P3:LB6, VB109
AENO
MOVB   #P4:LB7, VB110
LRD
MOVB   #P5:LB8, VB111
AENO
MOVB   #P6:LB9, VB112
AENO
MOVB   #P7:LB10, VB113
AENO
MOVB   #P8:LB11, VB114
LRD
MOVB   VB1029, VB115
AENO
MOVB   VB1030, VB116
AENO
MOVB   VB1031, VB117
AENO
MOVB   VB1032, VB118
AENO
MOVB   VB1033, VB119
LRD
MOVB   VB0, VB120
AENO
MOVB   VB0, VB121
LPP
MOVB   VB151, VB122
AENO
MOVB   VB152, VB123
AENO
MOVB   VB153, VB124
AENO
MOVB   VB154, VB125
AENO
MOVB   VB155, VB126
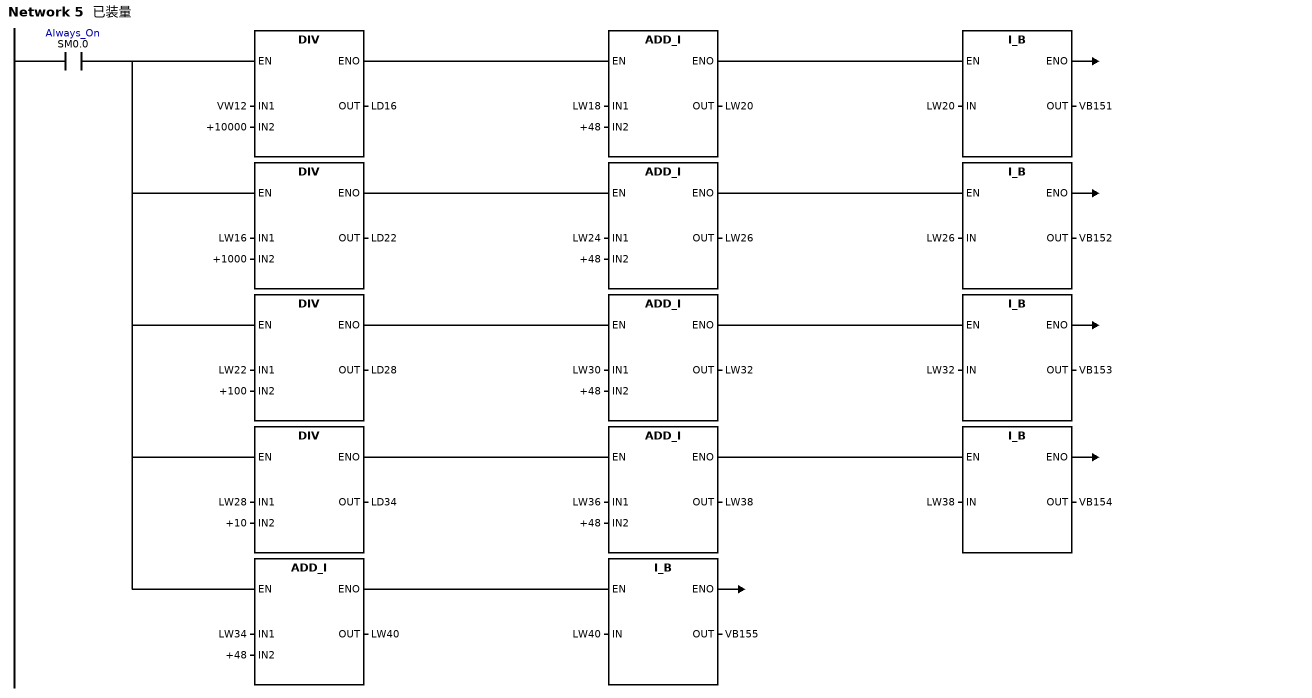
Network 5 // 已装量
LD     Always_On:SM0.0
LPS
MOVW   VW12, LW18
AENO
DIV    +10000, LD16
AENO
MOVW   LW18, LW20
AENO
+I     +48, LW20
AENO
ITB    LW20, VB151
LRD
MOVW   LW16, LW24
AENO
DIV    +1000, LD22
AENO
MOVW   LW24, LW26
AENO
+I     +48, LW26
AENO
ITB    LW26, VB152
LRD
MOVW   LW22, LW30
AENO
DIV    +100, LD28
AENO
MOVW   LW30, LW32
AENO
+I     +48, LW32
AENO
ITB    LW32, VB153
LRD
MOVW   LW28, LW36
AENO
DIV    +10, LD34
AENO
MOVW   LW36, LW38
AENO
+I     +48, LW38
AENO
ITB    LW38, VB154
LPP
MOVW   LW34, LW40
AENO
+I     +48, LW40
AENO
ITB    LW40, VB155
END_SUBROUTINE_BLOCK

SUBROUTINE_BLOCK LED2:SBR12
TITLE=
VAR_INPUT
D1:BYTE;	// LB0 
D2:BYTE;	// LB1 
D3:BYTE;	// LB2 
D4:BYTE;	// LB3 
P1:BYTE;	// LB4 
P2:BYTE;	// LB5 
P3:BYTE;	// LB6 
P4:BYTE;	// LB7 
P5:BYTE;	// LB8 
P6:BYTE;	// LB9 
P7:BYTE;	// LB10 
P8:BYTE;	// LB11 
RUN:WORD;	// LW12 
END_VAR
BEGIN
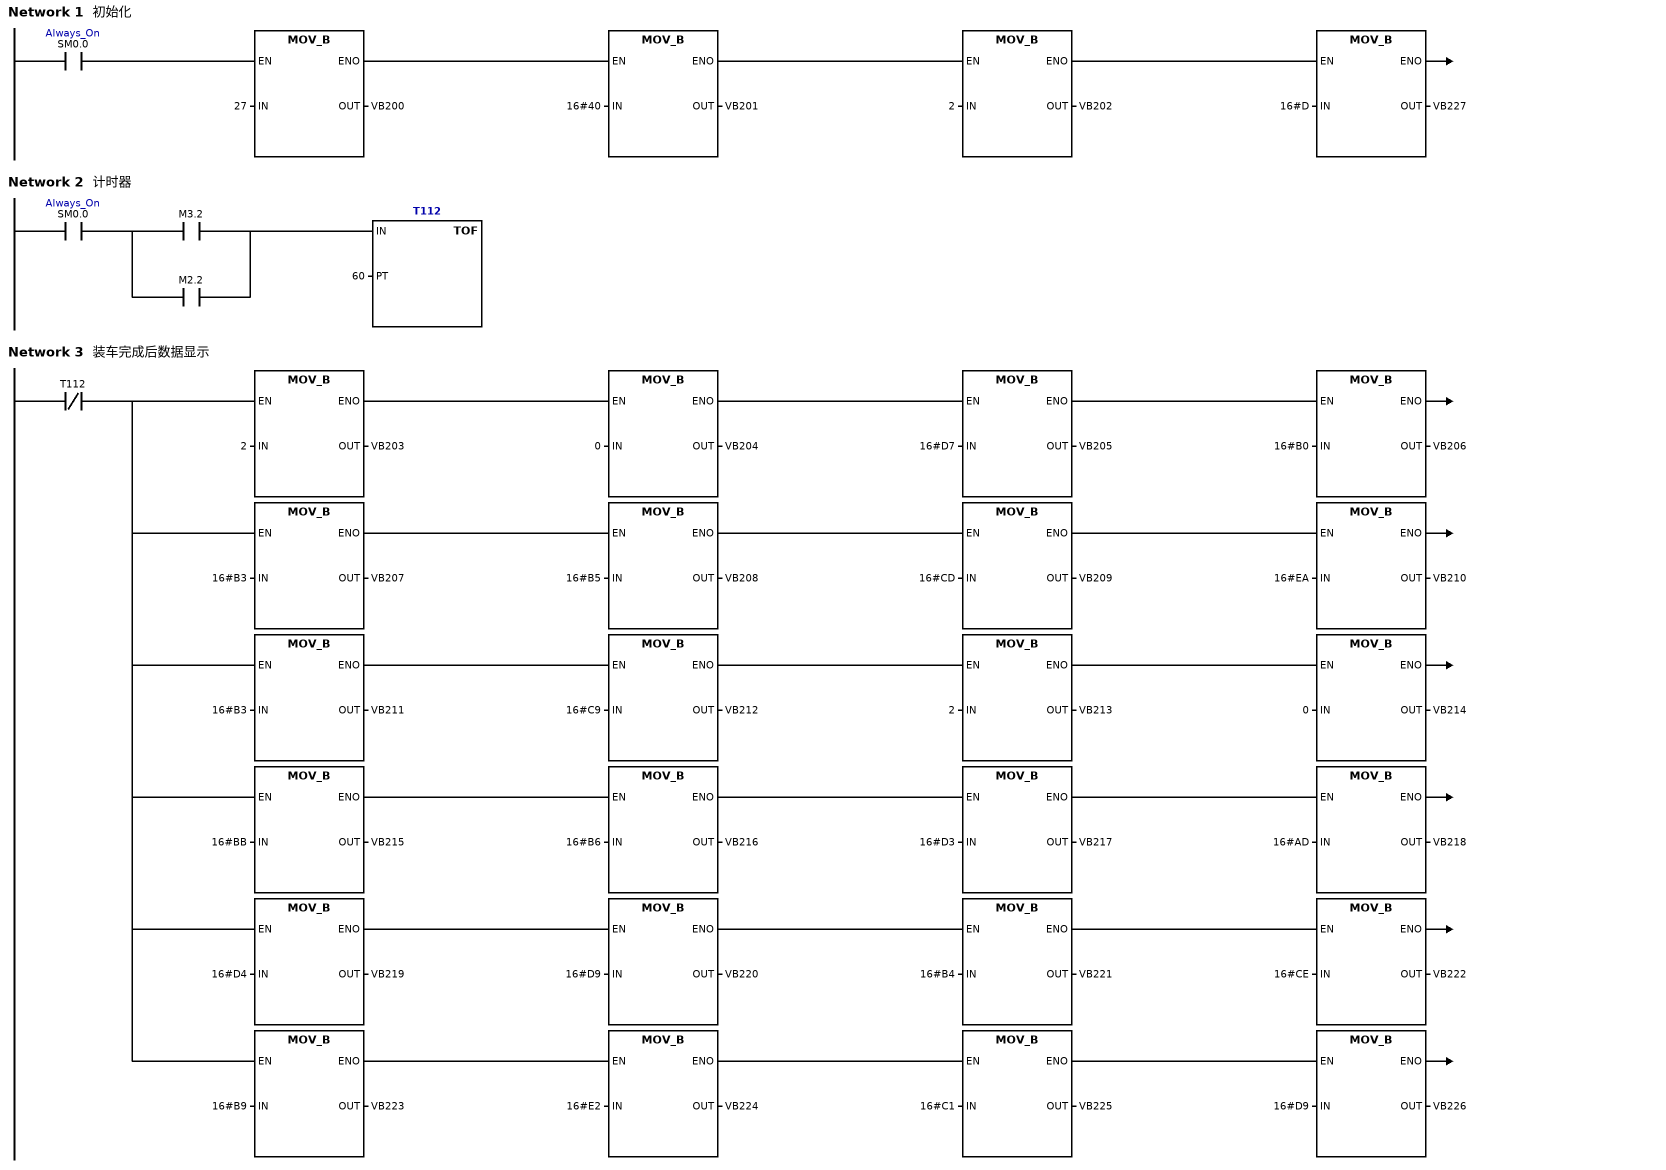
Network 1 // 初始化
LD     Always_On:SM0.0
MOVB   27, VB200
AENO
MOVB   16#40, VB201
AENO
MOVB   2, VB202
AENO
MOVB   16#D, VB227
Network 2 // 计时器
LD     Always_On:SM0.0
LD     M3.2
O      M2.2
ALD
TOF    T112, 60
Network 3 // 装车完成后数据显示
LDN    T112
LPS
MOVB   2, VB203
AENO
MOVB   0, VB204
AENO
MOVB   16#D7, VB205
AENO
MOVB   16#B0, VB206
LRD
MOVB   16#B3, VB207
AENO
MOVB   16#B5, VB208
AENO
MOVB   16#CD, VB209
AENO
MOVB   16#EA, VB210
LRD
MOVB   16#B3, VB211
AENO
MOVB   16#C9, VB212
AENO
MOVB   2, VB213
AENO
MOVB   0, VB214
LRD
MOVB   16#BB, VB215
AENO
MOVB   16#B6, VB216
AENO
MOVB   16#D3, VB217
AENO
MOVB   16#AD, VB218
LRD
MOVB   16#D4, VB219
AENO
MOVB   16#D9, VB220
AENO
MOVB   16#B4, VB221
AENO
MOVB   16#CE, VB222
LPP
MOVB   16#B9, VB223
AENO
MOVB   16#E2, VB224
AENO
MOVB   16#C1, VB225
AENO
MOVB   16#D9, VB226
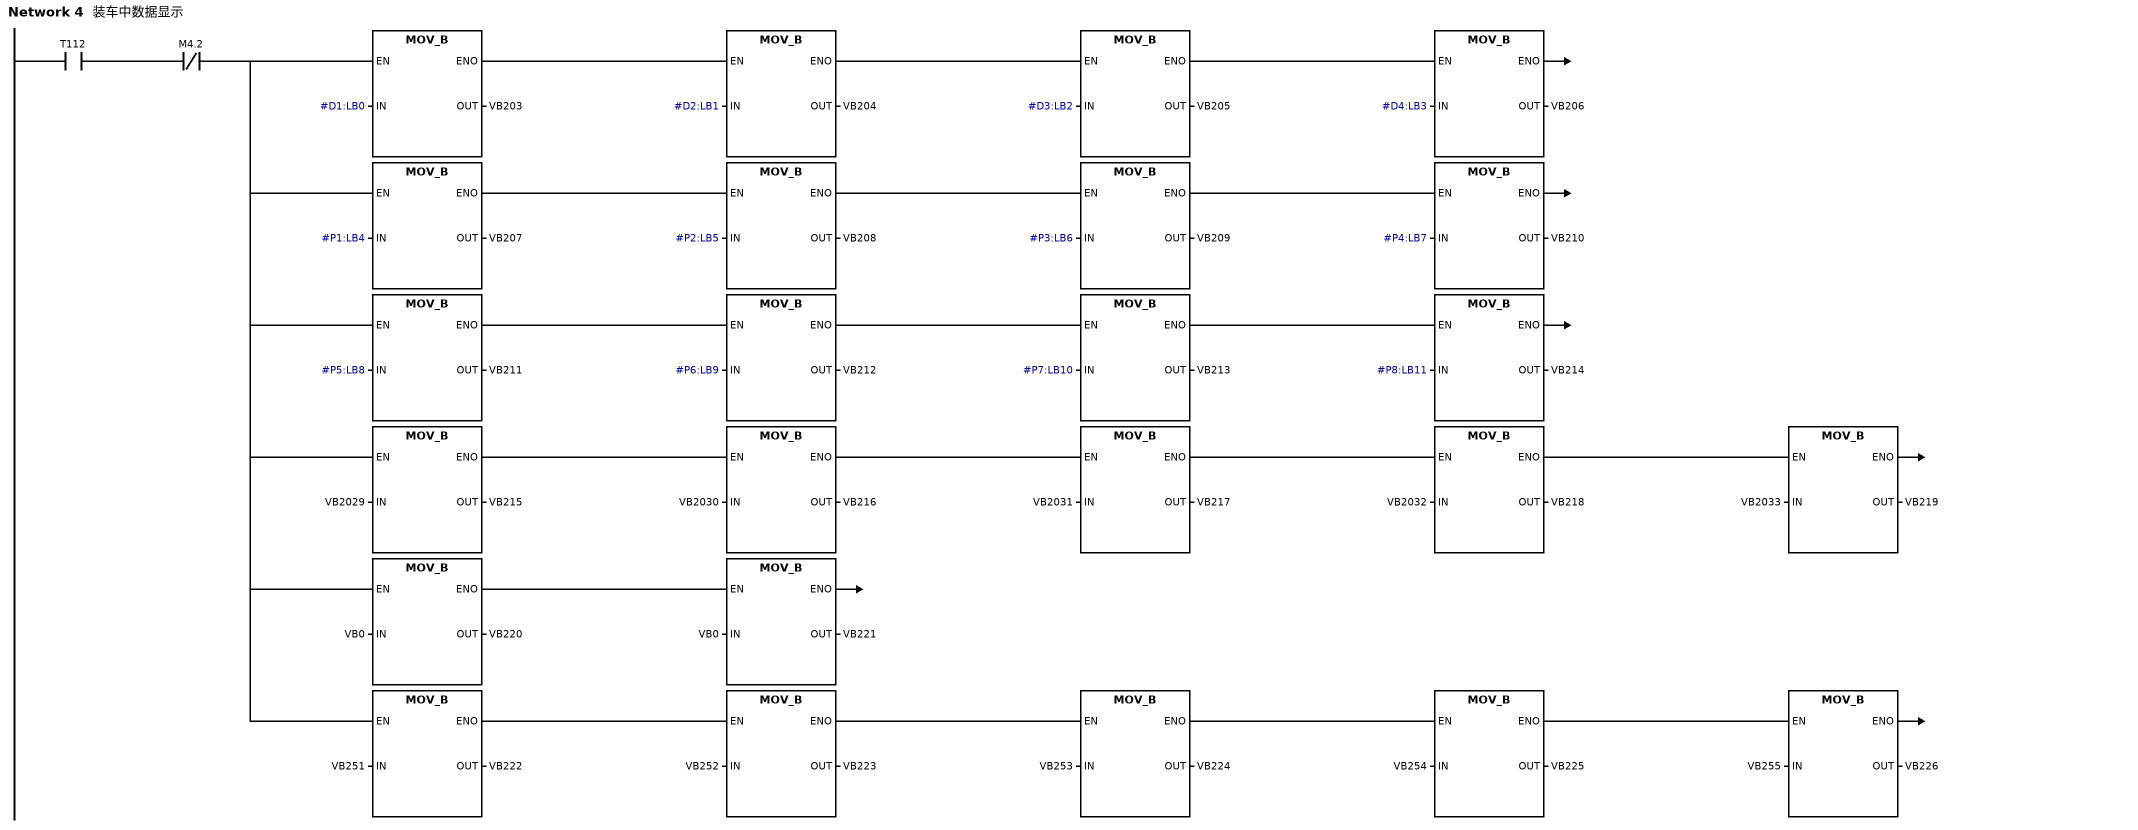
Network 4 // 装车中数据显示
LD     T112
AN     M4.2
LPS
MOVB   #D1:LB0, VB203
AENO
MOVB   #D2:LB1, VB204
AENO
MOVB   #D3:LB2, VB205
AENO
MOVB   #D4:LB3, VB206
LRD
MOVB   #P1:LB4, VB207
AENO
MOVB   #P2:LB5, VB208
AENO
MOVB   #P3:LB6, VB209
AENO
MOVB   #P4:LB7, VB210
LRD
MOVB   #P5:LB8, VB211
AENO
MOVB   #P6:LB9, VB212
AENO
MOVB   #P7:LB10, VB213
AENO
MOVB   #P8:LB11, VB214
LRD
MOVB   VB2029, VB215
AENO
MOVB   VB2030, VB216
AENO
MOVB   VB2031, VB217
AENO
MOVB   VB2032, VB218
AENO
MOVB   VB2033, VB219
LRD
MOVB   VB0, VB220
AENO
MOVB   VB0, VB221
LPP
MOVB   VB251, VB222
AENO
MOVB   VB252, VB223
AENO
MOVB   VB253, VB224
AENO
MOVB   VB254, VB225
AENO
MOVB   VB255, VB226
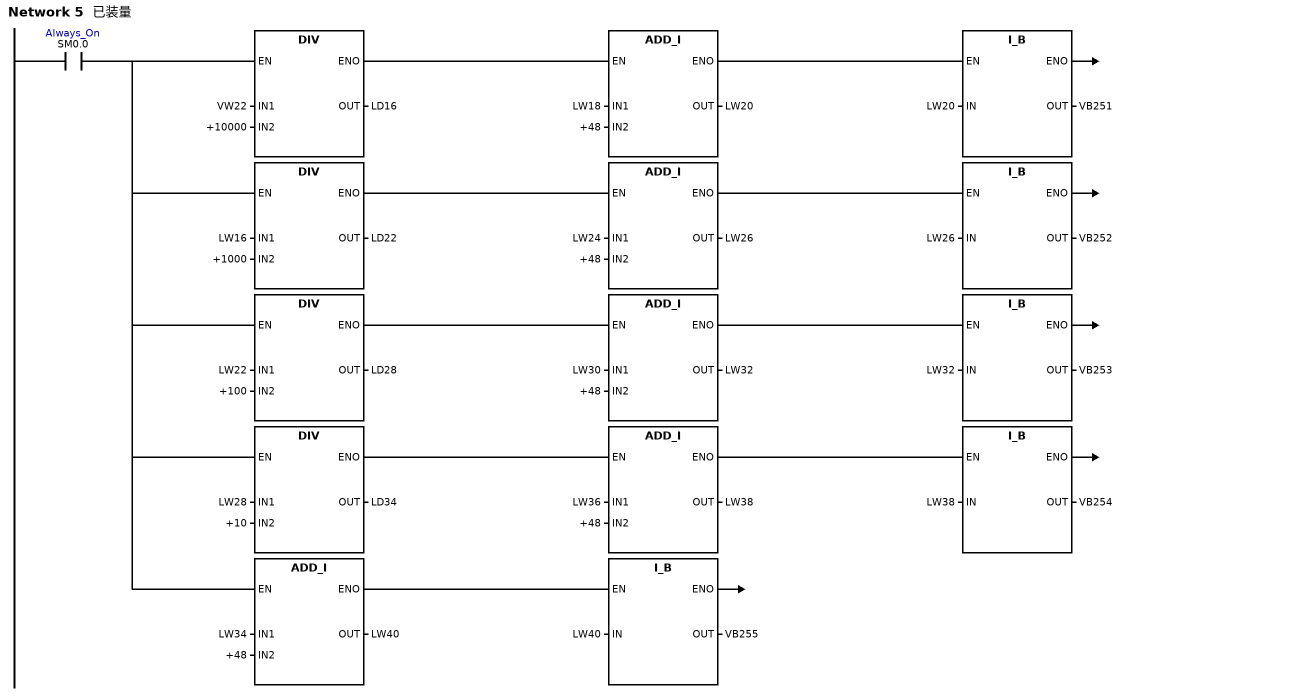
Network 5 // 已装量
LD     Always_On:SM0.0
LPS
MOVW   VW22, LW18
AENO
DIV    +10000, LD16
AENO
MOVW   LW18, LW20
AENO
+I     +48, LW20
AENO
ITB    LW20, VB251
LRD
MOVW   LW16, LW24
AENO
DIV    +1000, LD22
AENO
MOVW   LW24, LW26
AENO
+I     +48, LW26
AENO
ITB    LW26, VB252
LRD
MOVW   LW22, LW30
AENO
DIV    +100, LD28
AENO
MOVW   LW30, LW32
AENO
+I     +48, LW32
AENO
ITB    LW32, VB253
LRD
MOVW   LW28, LW36
AENO
DIV    +10, LD34
AENO
MOVW   LW36, LW38
AENO
+I     +48, LW38
AENO
ITB    LW38, VB254
LPP
MOVW   LW34, LW40
AENO
+I     +48, LW40
AENO
ITB    LW40, VB255
END_SUBROUTINE_BLOCK

SUBROUTINE_BLOCK LED3:SBR13
TITLE=
VAR_INPUT
D1:BYTE;	// LB0 
D2:BYTE;	// LB1 
D3:BYTE;	// LB2 
D4:BYTE;	// LB3 
P1:BYTE;	// LB4 
P2:BYTE;	// LB5 
P3:BYTE;	// LB6 
P4:BYTE;	// LB7 
P5:BYTE;	// LB8 
P6:BYTE;	// LB9 
P7:BYTE;	// LB10 
P8:BYTE;	// LB11 
RUN:WORD;	// LW12 
END_VAR
BEGIN
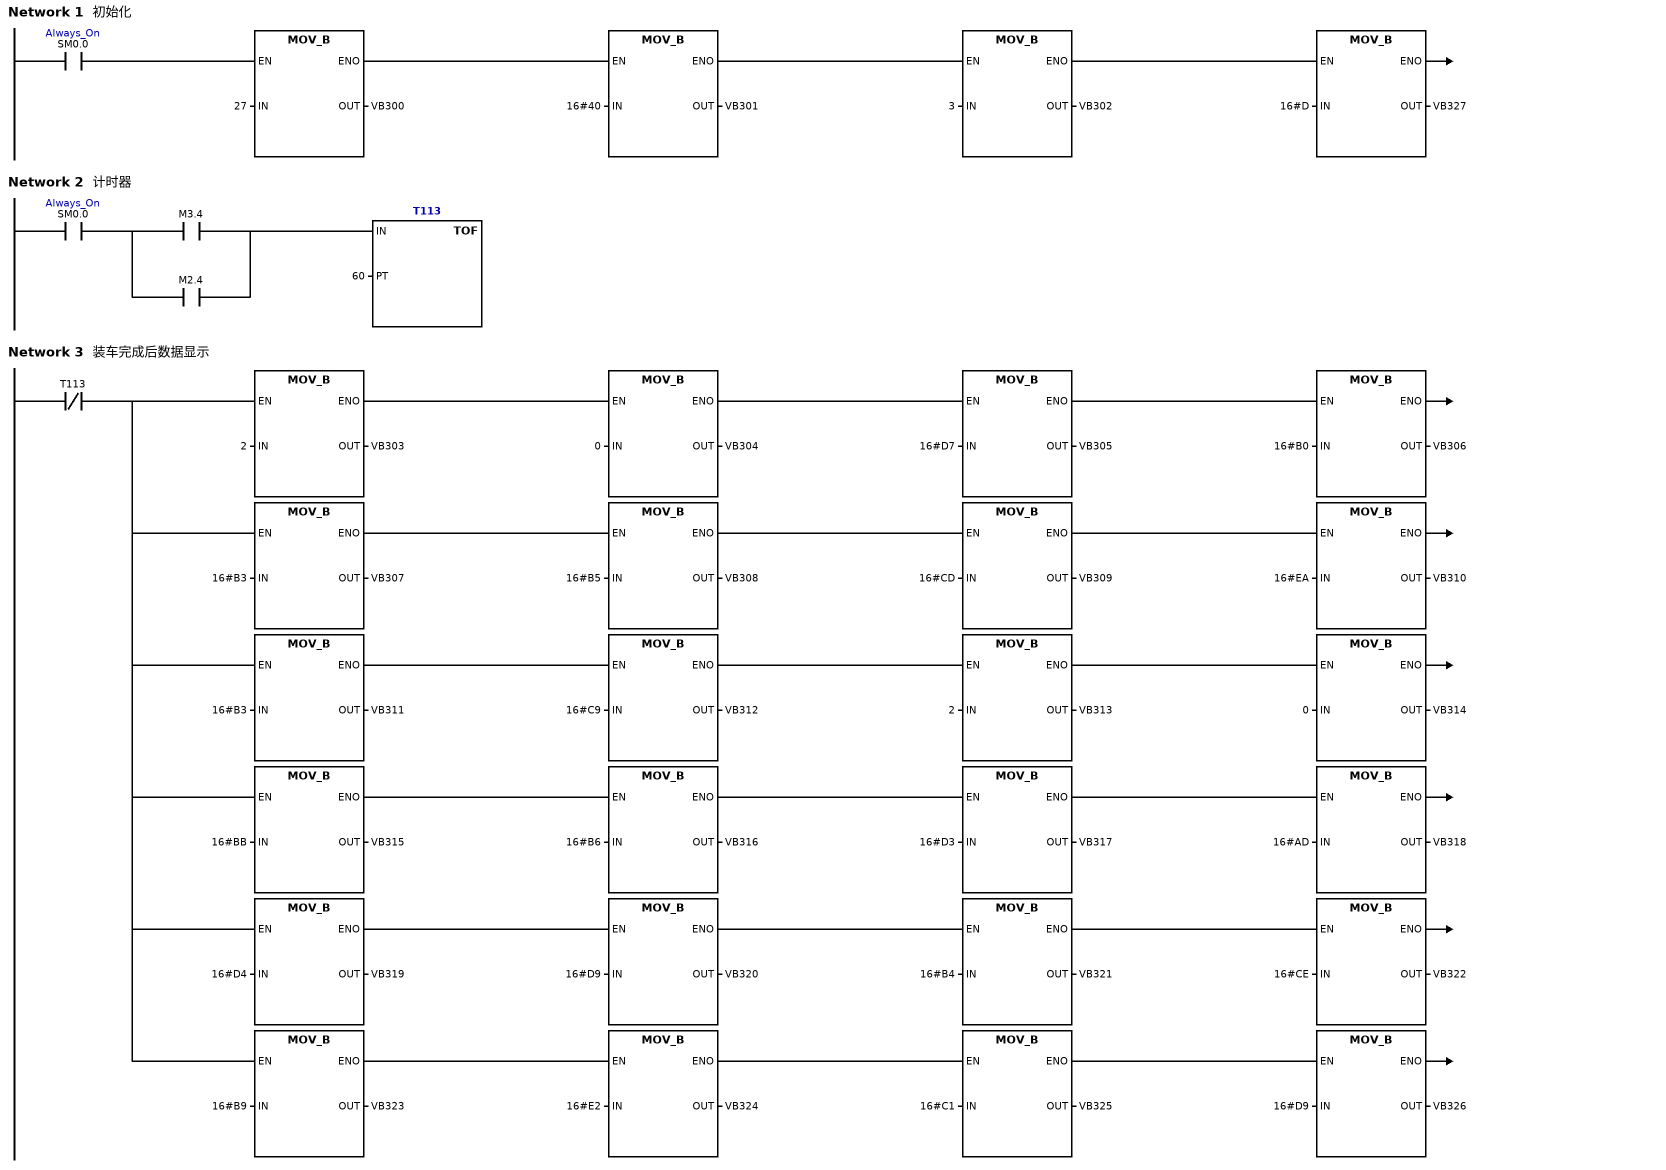
Network 1 // 初始化
LD     Always_On:SM0.0
MOVB   27, VB300
AENO
MOVB   16#40, VB301
AENO
MOVB   3, VB302
AENO
MOVB   16#D, VB327
Network 2 // 计时器
LD     Always_On:SM0.0
LD     M3.4
O      M2.4
ALD
TOF    T113, 60
Network 3 // 装车完成后数据显示
LDN    T113
LPS
MOVB   2, VB303
AENO
MOVB   0, VB304
AENO
MOVB   16#D7, VB305
AENO
MOVB   16#B0, VB306
LRD
MOVB   16#B3, VB307
AENO
MOVB   16#B5, VB308
AENO
MOVB   16#CD, VB309
AENO
MOVB   16#EA, VB310
LRD
MOVB   16#B3, VB311
AENO
MOVB   16#C9, VB312
AENO
MOVB   2, VB313
AENO
MOVB   0, VB314
LRD
MOVB   16#BB, VB315
AENO
MOVB   16#B6, VB316
AENO
MOVB   16#D3, VB317
AENO
MOVB   16#AD, VB318
LRD
MOVB   16#D4, VB319
AENO
MOVB   16#D9, VB320
AENO
MOVB   16#B4, VB321
AENO
MOVB   16#CE, VB322
LPP
MOVB   16#B9, VB323
AENO
MOVB   16#E2, VB324
AENO
MOVB   16#C1, VB325
AENO
MOVB   16#D9, VB326
